LIN {X 0,Y 370.068,Z 490.091,A -85,B 0,C 180,E1 -12871.089,E2 -12871.089} C_VEL
LIN {X 0,Y 369.236,Z 499.209,A -85,B 0,C 180,E1 -12872.728,E2 -12872.728} C_VEL
LIN {X 0,Y 368.632,Z 506.554,A -85,B 0,C 180,E1 -12874.374,E2 -12874.374} C_VEL
LIN {X 0,Y 368.208,Z 512.444,A -85,B 0,C 180,E1 -12876.027,E2 -12876.027} C_VEL
LIN {X 0,Y 367.86,Z 517.099,A -85,B 0,C 180,E1 -12877.686,E2 -12877.686} C_VEL
LIN {X 0,Y 367.581,Z 520.649,A -85,B 0,C 180,E1 -12879.354,E2 -12879.354} C_VEL
LIN {X 0,Y 367.418,Z 523.176,A -85,B 0,C 180,E1 -12881.028,E2 -12881.028} C_VEL
LIN {X 0,Y 367.364,Z 524.704,A -85,B 0,C 180,E1 -12882.662,E2 -12882.662} C_VEL
LIN {X 0,Y 367.283,Z 525.373,A -85,B 0,C 180,E1 -12884.405,E2 -12884.405} C_VEL
LIN {X 0,Y 367.336,Z 525.296,A -85,B 0,C 180,E1 -12885.537,E2 -12885.537} C_VEL
LIN {X 0,Y 367.455,Z 524.256,A -85,B 0,C 180,E1 -12887.304,E2 -12887.304} C_VEL
LIN {X 0,Y 367.684,Z 522.431,A -85,B 0,C 180,E1 -12888.963,E2 -12888.963} C_VEL
LIN {X 0,Y 368.051,Z 519.521,A -85,B 0,C 180,E1 -12890.664,E2 -12890.664} C_VEL
LIN {X 0,Y 368.43,Z 516.667,A -85,B 0,C 180,E1 -12891.919,E2 -12891.919} C_VEL
LIN {X 0,Y 368.033,Z 514.487,A -85,B 0,C 180,E1 -12892.771,E2 -12892.771} C_VEL
LIN {X 0,Y 365.711,Z 510.618,A -85,B 0,C 180,E1 -12894.153,E2 -12894.153} C_VEL
LIN {X 0,Y 363.521,Z 506.158,A -85,B 0,C 180,E1 -12895.502,E2 -12895.502} C_VEL
LIN {X 0,Y 363.329,Z 502.988,A -85,B 0,C 180,E1 -12896.289,E2 -12896.289} C_VEL
LIN {X 0,Y 364.425,Z 495.192,A -85,B 0,C 180,E1 -12897.883,E2 -12897.883} C_VEL
LIN {X 0,Y 365.532,Z 486.293,A -85,B 0,C 180,E1 -12899.36,E2 -12899.36} C_VEL
LIN {X 0,Y 366.817,Z 476.517,A -85,B 0,C 180,E1 -12900.658,E2 -12900.658} C_VEL
LIN {X 0,Y 368.109,Z 465.503,A -85,B 0,C 180,E1 -12901.832,E2 -12901.832} C_VEL
LIN {X 0,Y 369.097,Z 454.561,A -85,B 0,C 180,E1 -12902.761,E2 -12902.761} C_VEL
LIN {X 0,Y 370.067,Z 441.667,A -85,B 0,C 180,E1 -12903.582,E2 -12903.582} C_VEL
LIN {X 0,Y 370.776,Z 428.662,A -85,B 0,C 180,E1 -12904.163,E2 -12904.163} C_VEL
LIN {X 0,Y 371.143,Z 416.945,A -85,B 0,C 180,E1 -12904.494,E2 -12904.494} C_VEL
LIN {X 0,Y 372.737,Z 340.838,A -85,B 0,C 180,E1 -12905.987,E2 -12905.987} C_VEL
LIN {X 0,Y 369.659,Z 327.918,A -85,B 0,C 180,E1 -12906.496,E2 -12906.496} C_VEL
LIN {X 0,Y 364.062,Z 314.904,A -85,B 0,C 180,E1 -12907.224,E2 -12907.224} C_VEL
LIN {X 0,Y 361.901,Z 305.408,A -85,B 0,C 180,E1 -12909.94,E2 -12909.94} C_VEL
LIN {X 0,Y 361.838,Z 305.415,A -85,B 0,C 180,E1 -12912.829,E2 -12912.829} C_VEL
LIN {X 0,Y 361.82,Z 305.414,A -85,B 0,C 180,E1 -12915.947,E2 -12915.947} C_VEL
LIN {X 0,Y 361.838,Z 305.414,A -85,B 0,C 180,E1 -12919.244,E2 -12919.244} C_VEL
LIN {X 0,Y 361.866,Z 305.413,A -85,B 0,C 180,E1 -12922.777,E2 -12922.777} C_VEL
LIN {X 0,Y 361.856,Z 305.41,A -85,B 0,C 180,E1 -12925.72,E2 -12925.72} C_VEL
LIN {X 0,Y 361.876,Z 305.401,A -85,B 0,C 180,E1 -12929.672,E2 -12929.672} C_VEL
LIN {X 0,Y 361.956,Z 305.394,A -85,B 0,C 180,E1 -12933.475,E2 -12933.475} C_VEL
LIN {X 0,Y 361.891,Z 305.4,A -85,B 0,C 180,E1 -12937.145,E2 -12937.145} C_VEL
LIN {X 0,Y 361.922,Z 305.396,A -85,B 0,C 180,E1 -12940.724,E2 -12940.724} C_VEL
LIN {X 0,Y 361.947,Z 305.394,A -85,B 0,C 180,E1 -12944.226,E2 -12944.226} C_VEL
LIN {X 0,Y 362,Z 305.386,A -85,B 0,C 180,E1 -12946.528,E2 -12946.528} C_VEL
LIN {X 0,Y 362.032,Z 305.378,A -85,B 0,C 180,E1 -12949.938,E2 -12949.938} C_VEL
LIN {X 0,Y 362.151,Z 305.373,A -85,B 0,C 180,E1 -12952.192,E2 -12952.192} C_VEL
LIN {X 0,Y 362.117,Z 305.372,A -85,B 0,C 180,E1 -12954.431,E2 -12954.431} C_VEL
LIN {X 0,Y 362.281,Z 305.356,A -85,B 0,C 180,E1 -12957.776,E2 -12957.776} C_VEL
LIN {X 0,Y 362.426,Z 305.33,A -85,B 0,C 180,E1 -12960,E2 -12960} C_VEL
LIN {X 0,Y 362.281,Z 305.352,A -85,B 0,C 180,E1 -12962.224,E2 -12962.224} C_VEL
LIN {X 0,Y 362.171,Z 305.362,A -85,B 0,C 180,E1 -12966.686,E2 -12966.686} C_VEL
LIN {X 0,Y 362.075,Z 305.379,A -85,B 0,C 180,E1 -12968.933,E2 -12968.933} C_VEL
LIN {X 0,Y 361.96,Z 305.389,A -85,B 0,C 180,E1 -12972.332,E2 -12972.332} C_VEL
LIN {X 0,Y 361.963,Z 305.393,A -85,B 0,C 180,E1 -12974.62,E2 -12974.62} C_VEL
LIN {X 0,Y 361.961,Z 305.394,A -85,B 0,C 180,E1 -12978.099,E2 -12978.099} C_VEL
LIN {X 0,Y 361.863,Z 305.401,A -85,B 0,C 180,E1 -12981.655,E2 -12981.655} C_VEL
LIN {X 0,Y 361.928,Z 305.392,A -85,B 0,C 180,E1 -12985.29,E2 -12985.29} C_VEL
LIN {X 0,Y 361.919,Z 305.4,A -85,B 0,C 180,E1 -12987.778,E2 -12987.778} C_VEL
LIN {X 0,Y 361.848,Z 305.412,A -85,B 0,C 180,E1 -12991.285,E2 -12991.285} C_VEL
LIN {X 0,Y 361.855,Z 305.402,A -85,B 0,C 180,E1 -12994.28,E2 -12994.28} C_VEL
LIN {X 0,Y 361.864,Z 305.406,A -85,B 0,C 180,E1 -12997.223,E2 -12997.223} C_VEL
LIN {X 0,Y 361.837,Z 305.409,A -85,B 0,C 180,E1 -13000.755,E2 -13000.755} C_VEL
LIN {X 0,Y 361.819,Z 305.414,A -85,B 0,C 180,E1 -13004.368,E2 -13004.368} C_VEL
LIN {X 0,Y 361.838,Z 305.413,A -85,B 0,C 180,E1 -13007.568,E2 -13007.568} C_VEL
LIN {X 0,Y 361.87,Z 305.399,A -85,B 0,C 180,E1 -13010.974,E2 -13010.974} C_VEL
LIN {X 0,Y 361.876,Z 305.405,A -85,B 0,C 180,E1 -13014.655,E2 -13014.655} C_VEL
LIN {X 0,Y 361.937,Z 305.571,A -85,B 0,C 180,E1 -13018.542,E2 -13018.542} C_VEL
LIN {X 0,Y 364.825,Z 317.71,A -85,B 0,C 180,E1 -13021.834,E2 -13021.834} C_VEL
LIN {X 0,Y 366.693,Z 327.189,A -85,B 0,C 180,E1 -13024.263,E2 -13024.263} C_VEL
LIN {X 0,Y 365.539,Z 339.041,A -85,B 0,C 180,E1 -13026.955,E2 -13026.955} C_VEL
LIN {X 0,Y 369.976,Z 360.901,A -85,B 0,C 180,E1 -13027.767,E2 -13027.767} C_VEL
LIN {X 0,Y 372.124,Z 375.435,A -85,B 0,C 180,E1 -13028.232,E2 -13028.232} C_VEL
LIN {X 0,Y 370.71,Z 446.624,A -85,B 0,C 180,E1 -13029.649,E2 -13029.649} C_VEL
LIN {X 0,Y 370.056,Z 459.471,A -85,B 0,C 180,E1 -13030.082,E2 -13030.082} C_VEL
LIN {X 0,Y 369.035,Z 472.494,A -85,B 0,C 180,E1 -13030.749,E2 -13030.749} C_VEL
LIN {X 0,Y 367.885,Z 484.876,A -85,B 0,C 180,E1 -13031.626,E2 -13031.626} C_VEL
LIN {X 0,Y 366.487,Z 496.517,A -85,B 0,C 180,E1 -13032.708,E2 -13032.708} C_VEL
LIN {X 0,Y 365.196,Z 506.992,A -85,B 0,C 180,E1 -13033.94,E2 -13033.94} C_VEL
LIN {X 0,Y 364.106,Z 516.229,A -85,B 0,C 180,E1 -13035.287,E2 -13035.287} C_VEL
LIN {X 0,Y 362.967,Z 524.926,A -85,B 0,C 180,E1 -13036.849,E2 -13036.849} C_VEL
LIN {X 0,Y 361.882,Z 532.433,A -85,B 0,C 180,E1 -13038.517,E2 -13038.517} C_VEL
LIN {X 0,Y 361.11,Z 539.398,A -85,B 0,C 180,E1 -13040.477,E2 -13040.477} C_VEL
LIN {X 0,Y 360.68,Z 544.02,A -85,B 0,C 180,E1 -13042.16,E2 -13042.16} C_VEL
LIN {X 0,Y 360.424,Z 547.785,A -85,B 0,C 180,E1 -13043.969,E2 -13043.969} C_VEL
LIN {X 0,Y 360.366,Z 550.094,A -85,B 0,C 180,E1 -13045.525,E2 -13045.525} C_VEL
LIN {X 0,Y 360.301,Z 551.286,A -85,B 0,C 180,E1 -13046.645,E2 -13046.645} C_VEL
LIN {X 0,Y 360.358,Z 552.41,A -85,B 0,C 180,E1 -13048.882,E2 -13048.882} C_VEL
LIN {X 0,Y 360.423,Z 552.394,A -85,B 0,C 180,E1 -13049.999,E2 -13049.999} C_VEL
LIN {X 0,Y 360.389,Z 551.981,A -85,B 0,C 180,E1 -13051.117,E2 -13051.117} C_VEL
LIN {X 0,Y 360.327,Z 551.127,A -85,B 0,C 180,E1 -13052.235,E2 -13052.235} C_VEL
LIN {X 0,Y 360.322,Z 549.868,A -85,B 0,C 180,E1 -13053.354,E2 -13053.354} C_VEL
LIN {X 0,Y 360.375,Z 547.185,A -85,B 0,C 180,E1 -13055.034,E2 -13055.034} C_VEL
LIN {X 0,Y 360.497,Z 543.466,A -85,B 0,C 180,E1 -13056.716,E2 -13056.716} C_VEL
LIN {X 0,Y 360.741,Z 538.61,A -85,B 0,C 180,E1 -13058.401,E2 -13058.401} C_VEL
LIN {X 0,Y 361.155,Z 532.469,A -85,B 0,C 180,E1 -13060.086,E2 -13060.086} C_VEL
LIN {X 0,Y 361.774,Z 524.821,A -85,B 0,C 180,E1 -13061.769,E2 -13061.769} C_VEL
LIN {X 0,Y 362.468,Z 516.989,A -85,B 0,C 180,E1 -13063.168,E2 -13063.168} C_VEL
LIN {X 0,Y 363.389,Z 507.414,A -85,B 0,C 180,E1 -13064.561,E2 -13064.561} C_VEL
LIN {X 0,Y 364.251,Z 496.765,A -85,B 0,C 180,E1 -13065.814,E2 -13065.814} C_VEL
LIN {X 0,Y 365.096,Z 486.509,A -85,B 0,C 180,E1 -13066.782,E2 -13066.782} C_VEL
LIN {X 0,Y 366.026,Z 474.401,A -85,B 0,C 180,E1 -13067.674,E2 -13067.674} C_VEL
LIN {X 0,Y 366.831,Z 460.902,A -85,B 0,C 180,E1 -13068.391,E2 -13068.391} C_VEL
LIN {X 0,Y 367.36,Z 448.461,A -85,B 0,C 180,E1 -13068.834,E2 -13068.834} C_VEL
LIN {X 0,Y 368.505,Z 373.288,A -85,B 0,C 180,E1 -13070.322,E2 -13070.322} C_VEL
LIN {X 0,Y 363.871,Z 339.579,A -85,B 0,C 180,E1 -13071.257,E2 -13071.257} C_VEL
LIN {X 0,Y 365.148,Z 323.753,A -85,B 0,C 180,E1 -13074.746,E2 -13074.746} C_VEL
LIN {X 0,Y 364.78,Z 319.672,A -85,B 0,C 180,E1 -13075.692,E2 -13075.692} C_VEL
LIN {X 0,Y 362.332,Z 307.298,A -85,B 0,C 180,E1 -13078.688,E2 -13078.688} C_VEL
LIN {X 0,Y 361.932,Z 305.404,A -85,B 0,C 180,E1 -13079.184,E2 -13079.184} C_VEL
LIN {X 0,Y 361.857,Z 305.407,A -85,B 0,C 180,E1 -13083.369,E2 -13083.369} C_VEL
LIN {X 0,Y 361.863,Z 305.406,A -85,B 0,C 180,E1 -13087.017,E2 -13087.017} C_VEL
LIN {X 0,Y 361.85,Z 305.409,A -85,B 0,C 180,E1 -13089.86,E2 -13089.86} C_VEL
LIN {X 0,Y 361.831,Z 305.412,A -85,B 0,C 180,E1 -13092.828,E2 -13092.828} C_VEL
LIN {X 0,Y 361.814,Z 305.413,A -85,B 0,C 180,E1 -13095.945,E2 -13095.945} C_VEL
LIN {X 0,Y 361.831,Z 305.41,A -85,B 0,C 180,E1 -13099.243,E2 -13099.243} C_VEL
LIN {X 0,Y 361.865,Z 305.411,A -85,B 0,C 180,E1 -13102.775,E2 -13102.775} C_VEL
LIN {X 0,Y 361.849,Z 305.407,A -85,B 0,C 180,E1 -13105.719,E2 -13105.719} C_VEL
LIN {X 0,Y 361.87,Z 305.405,A -85,B 0,C 180,E1 -13109.672,E2 -13109.672} C_VEL
LIN {X 0,Y 361.947,Z 305.397,A -85,B 0,C 180,E1 -13113.474,E2 -13113.474} C_VEL
LIN {X 0,Y 361.882,Z 305.409,A -85,B 0,C 180,E1 -13117.144,E2 -13117.144} C_VEL
LIN {X 0,Y 361.898,Z 305.404,A -85,B 0,C 180,E1 -13120.723,E2 -13120.723} C_VEL
LIN {X 0,Y 361.924,Z 305.403,A -85,B 0,C 180,E1 -13123.066,E2 -13123.066} C_VEL
LIN {X 0,Y 361.99,Z 305.39,A -85,B 0,C 180,E1 -13126.527,E2 -13126.527} C_VEL
LIN {X 0,Y 362.023,Z 305.387,A -85,B 0,C 180,E1 -13129.938,E2 -13129.938} C_VEL
LIN {X 0,Y 362.142,Z 305.371,A -85,B 0,C 180,E1 -13132.192,E2 -13132.192} C_VEL
LIN {X 0,Y 362.108,Z 305.375,A -85,B 0,C 180,E1 -13134.431,E2 -13134.431} C_VEL
LIN {X 0,Y 362.273,Z 305.36,A -85,B 0,C 180,E1 -13137.776,E2 -13137.776} C_VEL
LIN {X 0,Y 362.418,Z 305.34,A -85,B 0,C 180,E1 -13140,E2 -13140} C_VEL
LIN {X 0,Y 362.274,Z 305.356,A -85,B 0,C 180,E1 -13142.224,E2 -13142.224} C_VEL
LIN {X 0,Y 362.126,Z 305.373,A -85,B 0,C 180,E1 -13146.687,E2 -13146.687} C_VEL
LIN {X 0,Y 362.022,Z 305.391,A -85,B 0,C 180,E1 -13150.062,E2 -13150.062} C_VEL
LIN {X 0,Y 361.989,Z 305.395,A -85,B 0,C 180,E1 -13153.899,E2 -13153.899} C_VEL
LIN {X 0,Y 361.959,Z 305.398,A -85,B 0,C 180,E1 -13157.939,E2 -13157.939} C_VEL
LIN {X 0,Y 361.853,Z 305.408,A -85,B 0,C 180,E1 -13161.656,E2 -13161.656} C_VEL
LIN {X 0,Y 361.918,Z 305.399,A -85,B 0,C 180,E1 -13165.291,E2 -13165.291} C_VEL
LIN {X 0,Y 361.91,Z 305.401,A -85,B 0,C 180,E1 -13167.779,E2 -13167.779} C_VEL
LIN {X 0,Y 361.839,Z 305.409,A -85,B 0,C 180,E1 -13171.286,E2 -13171.286} C_VEL
LIN {X 0,Y 361.847,Z 305.411,A -85,B 0,C 180,E1 -13174.281,E2 -13174.281} C_VEL
LIN {X 0,Y 361.853,Z 305.408,A -85,B 0,C 180,E1 -13177.223,E2 -13177.223} C_VEL
LIN {X 0,Y 361.807,Z 305.42,A -85,B 0,C 180,E1 -13180.752,E2 -13180.752} C_VEL
LIN {X 0,Y 361.811,Z 305.414,A -85,B 0,C 180,E1 -13184.37,E2 -13184.37} C_VEL
LIN {X 0,Y 361.825,Z 305.411,A -85,B 0,C 180,E1 -13187.57,E2 -13187.57} C_VEL
LIN {X 0,Y 361.84,Z 305.41,A -85,B 0,C 180,E1 -13191.573,E2 -13191.573} C_VEL
LIN {X 0,Y 361.871,Z 305.407,A -85,B 0,C 180,E1 -13194.657,E2 -13194.657} C_VEL
LIN {X 0,Y 361.835,Z 305.409,A -85,B 0,C 180,E1 -13198.372,E2 -13198.372} C_VEL
LIN {X 0,Y 361.864,Z 305.409,A -85,B 0,C 180,E1 -13200.953,E2 -13200.953} C_VEL
LIN {X 0,Y 361.872,Z 305.405,A -85,B 0,C 180,E1 -13204.707,E2 -13204.707} C_VEL
LIN {X 0,Y 361.86,Z 305.406,A -85,B 0,C 180,E1 -13208.346,E2 -13208.346} C_VEL
LIN {X 0,Y 361.92,Z 305.4,A -85,B 0,C 180,E1 -13212.086,E2 -13212.086} C_VEL
LIN {X 0,Y 361.962,Z 305.397,A -85,B 0,C 180,E1 -13215.381,E2 -13215.381} C_VEL
LIN {X 0,Y 361.961,Z 305.393,A -85,B 0,C 180,E1 -13218.805,E2 -13218.805} C_VEL
LIN {X 0,Y 362.053,Z 305.471,A -85,B 0,C 180,E1 -13220.469,E2 -13220.469} C_VEL
LIN {X 0,Y 363.779,Z 314.771,A -85,B 0,C 180,E1 -13222.852,E2 -13222.852} C_VEL
LIN {X 0,Y 365.738,Z 322.475,A -85,B 0,C 180,E1 -13223.108,E2 -13223.108} C_VEL
LIN {X 0,Y 368.937,Z 339.786,A -85,B 0,C 180,E1 -13223.615,E2 -13223.615} C_VEL
LIN {X 0,Y 367.596,Z 422.045,A -85,B 0,C 180,E1 -13225.237,E2 -13225.237} C_VEL
LIN {X 0,Y 367.117,Z 434.922,A -85,B 0,C 180,E1 -13225.701,E2 -13225.701} C_VEL
LIN {X 0,Y 366.581,Z 446.845,A -85,B 0,C 180,E1 -13226.337,E2 -13226.337} C_VEL
LIN {X 0,Y 365.927,Z 457.563,A -85,B 0,C 180,E1 -13227.097,E2 -13227.097} C_VEL
LIN {X 0,Y 365.136,Z 468.372,A -85,B 0,C 180,E1 -13228.071,E2 -13228.071} C_VEL
LIN {X 0,Y 364.2,Z 479.239,A -85,B 0,C 180,E1 -13229.31,E2 -13229.31} C_VEL
LIN {X 0,Y 363.293,Z 488.125,A -85,B 0,C 180,E1 -13230.555,E2 -13230.555} C_VEL
LIN {X 0,Y 362.544,Z 496.267,A -85,B 0,C 180,E1 -13231.945,E2 -13231.945} C_VEL
LIN {X 0,Y 361.803,Z 504.264,A -85,B 0,C 180,E1 -13233.62,E2 -13233.62} C_VEL
LIN {X 0,Y 361.268,Z 509.686,A -85,B 0,C 180,E1 -13235.023,E2 -13235.023} C_VEL
LIN {X 0,Y 360.921,Z 515.054,A -85,B 0,C 180,E1 -13236.736,E2 -13236.736} C_VEL
LIN {X 0,Y 360.632,Z 519.113,A -85,B 0,C 180,E1 -13238.405,E2 -13238.405} C_VEL
LIN {X 0,Y 360.37,Z 522.189,A -85,B 0,C 180,E1 -13240.11,E2 -13240.11} C_VEL
LIN {X 0,Y 360.33,Z 523.691,A -85,B 0,C 180,E1 -13241.248,E2 -13241.248} C_VEL
LIN {X 0,Y 360.265,Z 524.995,A -85,B 0,C 180,E1 -13242.736,E2 -13242.736} C_VEL
LIN {X 0,Y 360.212,Z 525.671,A -85,B 0,C 180,E1 -13244.694,E2 -13244.694} C_VEL
LIN {X 0,Y 360.259,Z 525.482,A -85,B 0,C 180,E1 -13245.85,E2 -13245.85} C_VEL
LIN {X 0,Y 360.358,Z 524.791,A -85,B 0,C 180,E1 -13247.129,E2 -13247.129} C_VEL
LIN {X 0,Y 360.482,Z 523.855,A -85,B 0,C 180,E1 -13248.177,E2 -13248.177} C_VEL
LIN {X 0,Y 360.667,Z 522.386,A -85,B 0,C 180,E1 -13249.346,E2 -13249.346} C_VEL
LIN {X 0,Y 361.022,Z 519.779,A -85,B 0,C 180,E1 -13250.866,E2 -13250.866} C_VEL
LIN {X 0,Y 361.659,Z 515.042,A -85,B 0,C 180,E1 -13252.871,E2 -13252.871} C_VEL
LIN {X 0,Y 362.568,Z 508.512,A -85,B 0,C 180,E1 -13254.916,E2 -13254.916} C_VEL
LIN {X 0,Y 363.329,Z 502.988,A -85,B 0,C 180,E1 -13256.289,E2 -13256.289} C_VEL
LIN {X 0,Y 363.141,Z 499.632,A -85,B 0,C 180,E1 -13257.058,E2 -13257.058} C_VEL
LIN {X 0,Y 361.072,Z 493.967,A -85,B 0,C 180,E1 -13258.31,E2 -13258.31} C_VEL
LIN {X 0,Y 359.182,Z 487.809,A -85,B 0,C 180,E1 -13259.501,E2 -13259.501} C_VEL
LIN {X 0,Y 359.253,Z 483.577,A -85,B 0,C 180,E1 -13260.16,E2 -13260.16} C_VEL
LIN {X 0,Y 360.561,Z 473.729,A -85,B 0,C 180,E1 -13261.413,E2 -13261.413} C_VEL
LIN {X 0,Y 361.9,Z 461.812,A -85,B 0,C 180,E1 -13262.609,E2 -13262.609} C_VEL
LIN {X 0,Y 362.944,Z 450.384,A -85,B 0,C 180,E1 -13263.503,E2 -13263.503} C_VEL
LIN {X 0,Y 363.793,Z 437.787,A -85,B 0,C 180,E1 -13264.24,E2 -13264.24} C_VEL
LIN {X 0,Y 364.457,Z 424.606,A -85,B 0,C 180,E1 -13264.755,E2 -13264.755} C_VEL
LIN {X 0,Y 365.042,Z 398.79,A -85,B 0,C 180,E1 -13265.32,E2 -13265.32} C_VEL
LIN {X 0,Y 366.313,Z 341.765,A -85,B 0,C 180,E1 -13266.456,E2 -13266.456} C_VEL
LIN {X 0,Y 363.572,Z 330.508,A -85,B 0,C 180,E1 -13266.92,E2 -13266.92} C_VEL
LIN {X 0,Y 356.907,Z 315.178,A -85,B 0,C 180,E1 -13267.82,E2 -13267.82} C_VEL
LIN {X 0,Y 354.827,Z 306.287,A -85,B 0,C 180,E1 -13270.451,E2 -13270.451} C_VEL
LIN {X 0,Y 354.769,Z 306.297,A -85,B 0,C 180,E1 -13273.896,E2 -13273.896} C_VEL
LIN {X 0,Y 354.797,Z 306.291,A -85,B 0,C 180,E1 -13277.663,E2 -13277.663} C_VEL
LIN {X 0,Y 354.817,Z 306.277,A -85,B 0,C 180,E1 -13280.666,E2 -13280.666} C_VEL
LIN {X 0,Y 354.824,Z 306.285,A -85,B 0,C 180,E1 -13284.301,E2 -13284.301} C_VEL
LIN {X 0,Y 354.788,Z 306.29,A -85,B 0,C 180,E1 -13287.667,E2 -13287.667} C_VEL
LIN {X 0,Y 354.871,Z 306.276,A -85,B 0,C 180,E1 -13290.621,E2 -13290.621} C_VEL
LIN {X 0,Y 354.901,Z 306.273,A -85,B 0,C 180,E1 -13294.173,E2 -13294.173} C_VEL
LIN {X 0,Y 354.836,Z 306.282,A -85,B 0,C 180,E1 -13297.894,E2 -13297.894} C_VEL
LIN {X 0,Y 354.924,Z 306.27,A -85,B 0,C 180,E1 -13301.891,E2 -13301.891} C_VEL
LIN {X 0,Y 354.944,Z 306.264,A -85,B 0,C 180,E1 -13305.981,E2 -13305.981} C_VEL
LIN {X 0,Y 354.979,Z 306.259,A -85,B 0,C 180,E1 -13309.736,E2 -13309.736} C_VEL
LIN {X 0,Y 355.114,Z 306.25,A -85,B 0,C 180,E1 -13312.037,E2 -13312.037} C_VEL
LIN {X 0,Y 355.091,Z 306.247,A -85,B 0,C 180,E1 -13314.321,E2 -13314.321} C_VEL
LIN {X 0,Y 355.244,Z 306.232,A -85,B 0,C 180,E1 -13317.732,E2 -13317.732} C_VEL
LIN {X 0,Y 355.375,Z 306.208,A -85,B 0,C 180,E1 -13320,E2 -13320} C_VEL
LIN {X 0,Y 355.244,Z 306.229,A -85,B 0,C 180,E1 -13322.268,E2 -13322.268} C_VEL
LIN {X 0,Y 355.137,Z 306.239,A -85,B 0,C 180,E1 -13326.819,E2 -13326.819} C_VEL
LIN {X 0,Y 355.016,Z 306.258,A -85,B 0,C 180,E1 -13329.112,E2 -13329.112} C_VEL
LIN {X 0,Y 354.921,Z 306.27,A -85,B 0,C 180,E1 -13332.581,E2 -13332.581} C_VEL
LIN {X 0,Y 354.89,Z 306.269,A -85,B 0,C 180,E1 -13336.096,E2 -13336.096} C_VEL
LIN {X 0,Y 354.908,Z 306.276,A -85,B 0,C 180,E1 -13338.472,E2 -13338.472} C_VEL
LIN {X 0,Y 354.818,Z 306.28,A -85,B 0,C 180,E1 -13342.107,E2 -13342.107} C_VEL
LIN {X 0,Y 354.9,Z 306.265,A -85,B 0,C 180,E1 -13345.827,E2 -13345.827} C_VEL
LIN {X 0,Y 354.855,Z 306.272,A -85,B 0,C 180,E1 -13349.678,E2 -13349.678} C_VEL
LIN {X 0,Y 354.808,Z 306.28,A -85,B 0,C 180,E1 -13353.702,E2 -13353.702} C_VEL
LIN {X 0,Y 354.799,Z 306.288,A -85,B 0,C 180,E1 -13356.459,E2 -13356.459} C_VEL
LIN {X 0,Y 354.826,Z 306.286,A -85,B 0,C 180,E1 -13359.424,E2 -13359.424} C_VEL
LIN {X 0,Y 354.79,Z 306.291,A -85,B 0,C 180,E1 -13362.867,E2 -13362.867} C_VEL
LIN {X 0,Y 354.768,Z 306.292,A -85,B 0,C 180,E1 -13366.103,E2 -13366.103} C_VEL
LIN {X 0,Y 354.79,Z 306.293,A -85,B 0,C 180,E1 -13369.179,E2 -13369.179} C_VEL
LIN {X 0,Y 354.809,Z 306.291,A -85,B 0,C 180,E1 -13372.403,E2 -13372.403} C_VEL
LIN {X 0,Y 354.814,Z 306.286,A -85,B 0,C 180,E1 -13374.941,E2 -13374.941} C_VEL
LIN {X 0,Y 354.869,Z 306.451,A -85,B 0,C 180,E1 -13378.035,E2 -13378.035} C_VEL
LIN {X 0,Y 357.633,Z 317.839,A -85,B 0,C 180,E1 -13381.219,E2 -13381.219} C_VEL
LIN {X 0,Y 359.745,Z 328.336,A -85,B 0,C 180,E1 -13383.983,E2 -13383.983} C_VEL
LIN {X 0,Y 359.604,Z 331.955,A -85,B 0,C 180,E1 -13384.844,E2 -13384.844} C_VEL
LIN {X 0,Y 358.872,Z 338.719,A -85,B 0,C 180,E1 -13386.404,E2 -13386.404} C_VEL
LIN {X 0,Y 363.562,Z 361.716,A -85,B 0,C 180,E1 -13387.296,E2 -13387.296} C_VEL
LIN {X 0,Y 365.709,Z 376.184,A -85,B 0,C 180,E1 -13387.775,E2 -13387.775} C_VEL
LIN {X 0,Y 364.171,Z 447.686,A -85,B 0,C 180,E1 -13389.23,E2 -13389.23} C_VEL
LIN {X 0,Y 363.369,Z 461.513,A -85,B 0,C 180,E1 -13389.737,E2 -13389.737} C_VEL
LIN {X 0,Y 362.271,Z 474.46,A -85,B 0,C 180,E1 -13390.448,E2 -13390.448} C_VEL
LIN {X 0,Y 360.966,Z 487,A -85,B 0,C 180,E1 -13391.408,E2 -13391.408} C_VEL
LIN {X 0,Y 359.541,Z 498.198,A -85,B 0,C 180,E1 -13392.51,E2 -13392.51} C_VEL
LIN {X 0,Y 358.236,Z 508.311,A -85,B 0,C 180,E1 -13393.765,E2 -13393.765} C_VEL
LIN {X 0,Y 357.068,Z 517.439,A -85,B 0,C 180,E1 -13395.174,E2 -13395.174} C_VEL
LIN {X 0,Y 355.84,Z 526.358,A -85,B 0,C 180,E1 -13396.871,E2 -13396.871} C_VEL
LIN {X 0,Y 354.753,Z 533.563,A -85,B 0,C 180,E1 -13398.573,E2 -13398.573} C_VEL
LIN {X 0,Y 354.071,Z 539.342,A -85,B 0,C 180,E1 -13400.286,E2 -13400.286} C_VEL
LIN {X 0,Y 353.624,Z 543.914,A -85,B 0,C 180,E1 -13402.002,E2 -13402.002} C_VEL
LIN {X 0,Y 353.318,Z 547.914,A -85,B 0,C 180,E1 -13404.029,E2 -13404.029} C_VEL
LIN {X 0,Y 353.279,Z 549.914,A -85,B 0,C 180,E1 -13405.435,E2 -13405.435} C_VEL
LIN {X 0,Y 353.223,Z 551.071,A -85,B 0,C 180,E1 -13406.577,E2 -13406.577} C_VEL
LIN {X 0,Y 353.259,Z 552.154,A -85,B 0,C 180,E1 -13408.859,E2 -13408.859} C_VEL
LIN {X 0,Y 353.328,Z 552.119,A -85,B 0,C 180,E1 -13409.999,E2 -13409.999} C_VEL
LIN {X 0,Y 353.292,Z 551.675,A -85,B 0,C 180,E1 -13411.139,E2 -13411.139} C_VEL
LIN {X 0,Y 353.243,Z 549.517,A -85,B 0,C 180,E1 -13413.421,E2 -13413.421} C_VEL
LIN {X 0,Y 353.278,Z 546.793,A -85,B 0,C 180,E1 -13415.135,E2 -13415.135} C_VEL
LIN {X 0,Y 353.415,Z 543.03,A -85,B 0,C 180,E1 -13416.852,E2 -13416.852} C_VEL
LIN {X 0,Y 353.679,Z 538.128,A -85,B 0,C 180,E1 -13418.57,E2 -13418.57} C_VEL
LIN {X 0,Y 354.12,Z 531.935,A -85,B 0,C 180,E1 -13420.288,E2 -13420.288} C_VEL
LIN {X 0,Y 354.801,Z 524.222,A -85,B 0,C 180,E1 -13422.003,E2 -13422.003} C_VEL
LIN {X 0,Y 355.506,Z 516.304,A -85,B 0,C 180,E1 -13423.431,E2 -13423.431} C_VEL
LIN {X 0,Y 356.437,Z 506.628,A -85,B 0,C 180,E1 -13424.851,E2 -13424.851} C_VEL
LIN {X 0,Y 357.355,Z 495.865,A -85,B 0,C 180,E1 -13426.127,E2 -13426.127} C_VEL
LIN {X 0,Y 358.235,Z 485.46,A -85,B 0,C 180,E1 -13427.113,E2 -13427.113} C_VEL
LIN {X 0,Y 359.229,Z 473.014,A -85,B 0,C 180,E1 -13428.019,E2 -13428.019} C_VEL
LIN {X 0,Y 360,Z 459.877,A -85,B 0,C 180,E1 -13428.716,E2 -13428.716} C_VEL
LIN {X 0,Y 360.627,Z 446.984,A -85,B 0,C 180,E1 -13429.162,E2 -13429.162} C_VEL
LIN {X 0,Y 361.661,Z 373.758,A -85,B 0,C 180,E1 -13430.633,E2 -13430.633} C_VEL
LIN {X 0,Y 356.94,Z 339.318,A -85,B 0,C 180,E1 -13431.611,E2 -13431.611} C_VEL
LIN {X 0,Y 358.184,Z 324.465,A -85,B 0,C 180,E1 -13434.951,E2 -13434.951} C_VEL
LIN {X 0,Y 357.448,Z 319.009,A -85,B 0,C 180,E1 -13436.255,E2 -13436.255} C_VEL
LIN {X 0,Y 354.876,Z 306.283,A -85,B 0,C 180,E1 -13439.431,E2 -13439.431} C_VEL
LIN {X 0,Y 354.803,Z 306.287,A -85,B 0,C 180,E1 -13443.701,E2 -13443.701} C_VEL
LIN {X 0,Y 354.794,Z 306.291,A -85,B 0,C 180,E1 -13446.458,E2 -13446.458} C_VEL
LIN {X 0,Y 354.82,Z 306.283,A -85,B 0,C 180,E1 -13449.422,E2 -13449.422} C_VEL
LIN {X 0,Y 354.783,Z 306.29,A -85,B 0,C 180,E1 -13452.866,E2 -13452.866} C_VEL
LIN {X 0,Y 354.763,Z 306.293,A -85,B 0,C 180,E1 -13456.103,E2 -13456.103} C_VEL
LIN {X 0,Y 354.783,Z 306.289,A -85,B 0,C 180,E1 -13459.178,E2 -13459.178} C_VEL
LIN {X 0,Y 354.806,Z 306.288,A -85,B 0,C 180,E1 -13462.401,E2 -13462.401} C_VEL
LIN {X 0,Y 354.806,Z 306.289,A -85,B 0,C 180,E1 -13464.94,E2 -13464.94} C_VEL
LIN {X 0,Y 354.808,Z 306.287,A -85,B 0,C 180,E1 -13468.398,E2 -13468.398} C_VEL
LIN {X 0,Y 354.847,Z 306.28,A -85,B 0,C 180,E1 -13471.619,E2 -13471.619} C_VEL
LIN {X 0,Y 354.891,Z 306.274,A -85,B 0,C 180,E1 -13474.172,E2 -13474.172} C_VEL
LIN {X 0,Y 354.826,Z 306.282,A -85,B 0,C 180,E1 -13477.893,E2 -13477.893} C_VEL
LIN {X 0,Y 354.914,Z 306.272,A -85,B 0,C 180,E1 -13481.891,E2 -13481.891} C_VEL
LIN {X 0,Y 354.934,Z 306.27,A -85,B 0,C 180,E1 -13485.981,E2 -13485.981} C_VEL
LIN {X 0,Y 354.969,Z 306.268,A -85,B 0,C 180,E1 -13489.736,E2 -13489.736} C_VEL
LIN {X 0,Y 355.105,Z 306.249,A -85,B 0,C 180,E1 -13492.037,E2 -13492.037} C_VEL
LIN {X 0,Y 355.083,Z 306.251,A -85,B 0,C 180,E1 -13494.321,E2 -13494.321} C_VEL
LIN {X 0,Y 355.236,Z 306.237,A -85,B 0,C 180,E1 -13497.732,E2 -13497.732} C_VEL
LIN {X 0,Y 355.388,Z 306.215,A -85,B 0,C 180,E1 -13500,E2 -13500} C_VEL
LIN {X 0,Y 355.237,Z 306.233,A -85,B 0,C 180,E1 -13502.268,E2 -13502.268} C_VEL
LIN {X 0,Y 355.09,Z 306.249,A -85,B 0,C 180,E1 -13506.82,E2 -13506.82} C_VEL
LIN {X 0,Y 354.969,Z 306.268,A -85,B 0,C 180,E1 -13510.264,E2 -13510.264} C_VEL
LIN {X 0,Y 354.934,Z 306.275,A -85,B 0,C 180,E1 -13514.019,E2 -13514.019} C_VEL
LIN {X 0,Y 354.915,Z 306.278,A -85,B 0,C 180,E1 -13518.109,E2 -13518.109} C_VEL
LIN {X 0,Y 354.807,Z 306.29,A -85,B 0,C 180,E1 -13522.108,E2 -13522.108} C_VEL
LIN {X 0,Y 354.89,Z 306.276,A -85,B 0,C 180,E1 -13525.828,E2 -13525.828} C_VEL
LIN {X 0,Y 354.847,Z 306.28,A -85,B 0,C 180,E1 -13529.679,E2 -13529.679} C_VEL
LIN {X 0,Y 354.8,Z 306.286,A -85,B 0,C 180,E1 -13533.703,E2 -13533.703} C_VEL
LIN {X 0,Y 354.79,Z 306.291,A -85,B 0,C 180,E1 -13536.461,E2 -13536.461} C_VEL
LIN {X 0,Y 354.762,Z 306.291,A -85,B 0,C 180,E1 -13539.414,E2 -13539.414} C_VEL
LIN {X 0,Y 354.78,Z 306.294,A -85,B 0,C 180,E1 -13542.868,E2 -13542.868} C_VEL
LIN {X 0,Y 354.761,Z 306.291,A -85,B 0,C 180,E1 -13546.105,E2 -13546.105} C_VEL
LIN {X 0,Y 354.761,Z 306.295,A -85,B 0,C 180,E1 -13549.177,E2 -13549.177} C_VEL
LIN {X 0,Y 354.797,Z 306.287,A -85,B 0,C 180,E1 -13552.405,E2 -13552.405} C_VEL
LIN {X 0,Y 354.809,Z 306.289,A -85,B 0,C 180,E1 -13554.942,E2 -13554.942} C_VEL
LIN {X 0,Y 354.79,Z 306.287,A -85,B 0,C 180,E1 -13558.406,E2 -13558.406} C_VEL
LIN {X 0,Y 354.794,Z 306.29,A -85,B 0,C 180,E1 -13561.615,E2 -13561.615} C_VEL
LIN {X 0,Y 354.839,Z 306.288,A -85,B 0,C 180,E1 -13565.423,E2 -13565.423} C_VEL
LIN {X 0,Y 354.826,Z 306.285,A -85,B 0,C 180,E1 -13569.114,E2 -13569.114} C_VEL
LIN {X 0,Y 354.88,Z 306.276,A -85,B 0,C 180,E1 -13572.72,E2 -13572.72} C_VEL
LIN {X 0,Y 354.952,Z 306.268,A -85,B 0,C 180,E1 -13576.256,E2 -13576.256} C_VEL
LIN {X 0,Y 355.015,Z 306.415,A -85,B 0,C 180,E1 -13580.242,E2 -13580.242} C_VEL
LIN {X 0,Y 356.578,Z 314.795,A -85,B 0,C 180,E1 -13582.481,E2 -13582.481} C_VEL
LIN {X 0,Y 358.947,Z 323.28,A -85,B 0,C 180,E1 -13582.782,E2 -13582.782} C_VEL
LIN {X 0,Y 362.173,Z 341.135,A -85,B 0,C 180,E1 -13583.315,E2 -13583.315} C_VEL
LIN {X 0,Y 360.763,Z 422.114,A -85,B 0,C 180,E1 -13584.937,E2 -13584.937} C_VEL
LIN {X 0,Y 360.264,Z 435.305,A -85,B 0,C 180,E1 -13585.42,E2 -13585.42} C_VEL
LIN {X 0,Y 359.673,Z 447.787,A -85,B 0,C 180,E1 -13586.104,E2 -13586.104} C_VEL
LIN {X 0,Y 358.934,Z 459.382,A -85,B 0,C 180,E1 -13586.963,E2 -13586.963} C_VEL
LIN {X 0,Y 358.056,Z 470.546,A -85,B 0,C 180,E1 -13588.032,E2 -13588.032} C_VEL
LIN {X 0,Y 357.072,Z 481.082,A -85,B 0,C 180,E1 -13589.296,E2 -13589.296} C_VEL
LIN {X 0,Y 356.178,Z 489.705,A -85,B 0,C 180,E1 -13590.566,E2 -13590.566} C_VEL
LIN {X 0,Y 355.43,Z 497.631,A -85,B 0,C 180,E1 -13591.984,E2 -13591.984} C_VEL
LIN {X 0,Y 354.708,Z 505.387,A -85,B 0,C 180,E1 -13593.693,E2 -13593.693} C_VEL
LIN {X 0,Y 354.166,Z 510.695,A -85,B 0,C 180,E1 -13595.124,E2 -13595.124} C_VEL
LIN {X 0,Y 353.836,Z 515.825,A -85,B 0,C 180,E1 -13596.845,E2 -13596.845} C_VEL
LIN {X 0,Y 353.533,Z 519.821,A -85,B 0,C 180,E1 -13598.575,E2 -13598.575} C_VEL
LIN {X 0,Y 353.259,Z 522.778,A -85,B 0,C 180,E1 -13600.315,E2 -13600.315} C_VEL
LIN {X 0,Y 353.215,Z 524.172,A -85,B 0,C 180,E1 -13601.478,E2 -13601.478} C_VEL
LIN {X 0,Y 353.176,Z 525.29,A -85,B 0,C 180,E1 -13602.819,E2 -13602.819} C_VEL
LIN {X 0,Y 353.117,Z 525.926,A -85,B 0,C 180,E1 -13604.996,E2 -13604.996} C_VEL
LIN {X 0,Y 353.294,Z 525.043,A -85,B 0,C 180,E1 -13607.281,E2 -13607.281} C_VEL
LIN {X 0,Y 353.461,Z 523.895,A -85,B 0,C 180,E1 -13608.551,E2 -13608.551} C_VEL
LIN {X 0,Y 353.829,Z 521.384,A -85,B 0,C 180,E1 -13610.341,E2 -13610.341} C_VEL
LIN {X 0,Y 354.372,Z 517.782,A -85,B 0,C 180,E1 -13612.137,E2 -13612.137} C_VEL
LIN {X 0,Y 355.011,Z 513.034,A -85,B 0,C 180,E1 -13613.918,E2 -13613.918} C_VEL
LIN {X 0,Y 355.922,Z 506.754,A -85,B 0,C 180,E1 -13615.748,E2 -13615.748} C_VEL
LIN {X 0,Y 356.983,Z 499.971,A -85,B 0,C 180,E1 -13617.328,E2 -13617.328} C_VEL
LIN {X 0,Y 358.23,Z 490.836,A -85,B 0,C 180,E1 -13619.05,E2 -13619.05} C_VEL
LIN {X 0,Y 359.253,Z 483.577,A -85,B 0,C 180,E1 -13620.16,E2 -13620.16} C_VEL
LIN {X 0,Y 359.36,Z 479.214,A -85,B 0,C 180,E1 -13620.796,E2 -13620.796} C_VEL
LIN {X 0,Y 357.636,Z 471.983,A -85,B 0,C 180,E1 -13621.85,E2 -13621.85} C_VEL
LIN {X 0,Y 355.771,Z 464.293,A -85,B 0,C 180,E1 -13622.813,E2 -13622.813} C_VEL
LIN {X 0,Y 355.64,Z 459.21,A -85,B 0,C 180,E1 -13623.298,E2 -13623.298} C_VEL
LIN {X 0,Y 356.68,Z 447.695,A -85,B 0,C 180,E1 -13624.15,E2 -13624.15} C_VEL
LIN {X 0,Y 357.534,Z 435.085,A -85,B 0,C 180,E1 -13624.84,E2 -13624.84} C_VEL
LIN {X 0,Y 358.119,Z 422.843,A -85,B 0,C 180,E1 -13625.29,E2 -13625.29} C_VEL
LIN {X 0,Y 360.004,Z 343.236,A -85,B 0,C 180,E1 -13626.928,E2 -13626.928} C_VEL
LIN {X 0,Y 357.634,Z 333.366,A -85,B 0,C 180,E1 -13627.343,E2 -13627.343} C_VEL
LIN {X 0,Y 349.749,Z 315.448,A -85,B 0,C 180,E1 -13628.449,E2 -13628.449} C_VEL
LIN {X 0,Y 347.771,Z 307.168,A -85,B 0,C 180,E1 -13630.933,E2 -13630.933} C_VEL
LIN {X 0,Y 347.725,Z 307.174,A -85,B 0,C 180,E1 -13633.408,E2 -13633.408} C_VEL
LIN {X 0,Y 347.727,Z 307.165,A -85,B 0,C 180,E1 -13636.686,E2 -13636.686} C_VEL
LIN {X 0,Y 347.749,Z 307.16,A -85,B 0,C 180,E1 -13640.173,E2 -13640.173} C_VEL
LIN {X 0,Y 347.764,Z 307.169,A -85,B 0,C 180,E1 -13642.679,E2 -13642.679} C_VEL
LIN {X 0,Y 347.75,Z 307.167,A -85,B 0,C 180,E1 -13645.956,E2 -13645.956} C_VEL
LIN {X 0,Y 347.766,Z 307.159,A -85,B 0,C 180,E1 -13649.653,E2 -13649.653} C_VEL
LIN {X 0,Y 347.853,Z 307.152,A -85,B 0,C 180,E1 -13652.745,E2 -13652.745} C_VEL
LIN {X 0,Y 347.79,Z 307.158,A -85,B 0,C 180,E1 -13656.162,E2 -13656.162} C_VEL
LIN {X 0,Y 347.819,Z 307.154,A -85,B 0,C 180,E1 -13659.91,E2 -13659.91} C_VEL
LIN {X 0,Y 347.868,Z 307.148,A -85,B 0,C 180,E1 -13662.359,E2 -13662.359} C_VEL
LIN {X 0,Y 347.899,Z 307.141,A -85,B 0,C 180,E1 -13665.971,E2 -13665.971} C_VEL
LIN {X 0,Y 347.929,Z 307.139,A -85,B 0,C 180,E1 -13669.526,E2 -13669.526} C_VEL
LIN {X 0,Y 348.106,Z 307.122,A -85,B 0,C 180,E1 -13673.042,E2 -13673.042} C_VEL
LIN {X 0,Y 348.206,Z 307.108,A -85,B 0,C 180,E1 -13677.686,E2 -13677.686} C_VEL
LIN {X 0,Y 348.325,Z 307.086,A -85,B 0,C 180,E1 -13680,E2 -13680} C_VEL
LIN {X 0,Y 348.207,Z 307.106,A -85,B 0,C 180,E1 -13682.313,E2 -13682.313} C_VEL
LIN {X 0,Y 348.105,Z 307.115,A -85,B 0,C 180,E1 -13686.958,E2 -13686.958} C_VEL
LIN {X 0,Y 347.929,Z 307.134,A -85,B 0,C 180,E1 -13690.474,E2 -13690.474} C_VEL
LIN {X 0,Y 347.9,Z 307.149,A -85,B 0,C 180,E1 -13694.15,E2 -13694.15} C_VEL
LIN {X 0,Y 347.893,Z 307.148,A -85,B 0,C 180,E1 -13698.29,E2 -13698.29} C_VEL
LIN {X 0,Y 347.769,Z 307.157,A -85,B 0,C 180,E1 -13701.626,E2 -13701.626} C_VEL
LIN {X 0,Y 347.812,Z 307.151,A -85,B 0,C 180,E1 -13705.108,E2 -13705.108} C_VEL
LIN {X 0,Y 347.812,Z 307.158,A -85,B 0,C 180,E1 -13707.694,E2 -13707.694} C_VEL
LIN {X 0,Y 347.765,Z 307.156,A -85,B 0,C 180,E1 -13710.346,E2 -13710.346} C_VEL
LIN {X 0,Y 347.746,Z 307.16,A -85,B 0,C 180,E1 -13714.464,E2 -13714.464} C_VEL
LIN {X 0,Y 347.775,Z 307.162,A -85,B 0,C 180,E1 -13717.988,E2 -13717.988} C_VEL
LIN {X 0,Y 347.752,Z 307.168,A -85,B 0,C 180,E1 -13721.83,E2 -13721.83} C_VEL
LIN {X 0,Y 347.708,Z 307.175,A -85,B 0,C 180,E1 -13725.027,E2 -13725.027} C_VEL
LIN {X 0,Y 347.752,Z 307.167,A -85,B 0,C 180,E1 -13728.397,E2 -13728.397} C_VEL
LIN {X 0,Y 347.775,Z 307.163,A -85,B 0,C 180,E1 -13732.011,E2 -13732.011} C_VEL
LIN {X 0,Y 347.747,Z 307.172,A -85,B 0,C 180,E1 -13735.536,E2 -13735.536} C_VEL
LIN {X 0,Y 347.775,Z 307.231,A -85,B 0,C 180,E1 -13737.471,E2 -13737.471} C_VEL
LIN {X 0,Y 350.73,Z 319.252,A -85,B 0,C 180,E1 -13740.926,E2 -13740.926} C_VEL
LIN {X 0,Y 352.811,Z 329.479,A -85,B 0,C 180,E1 -13743.689,E2 -13743.689} C_VEL
LIN {X 0,Y 352.938,Z 332.051,A -85,B 0,C 180,E1 -13744.335,E2 -13744.335} C_VEL
LIN {X 0,Y 352.185,Z 338.493,A -85,B 0,C 180,E1 -13745.845,E2 -13745.845} C_VEL
LIN {X 0,Y 357.073,Z 362.092,A -85,B 0,C 180,E1 -13746.787,E2 -13746.787} C_VEL
LIN {X 0,Y 359.319,Z 376.569,A -85,B 0,C 180,E1 -13747.289,E2 -13747.289} C_VEL
LIN {X 0,Y 357.787,Z 446.36,A -85,B 0,C 180,E1 -13748.728,E2 -13748.728} C_VEL
LIN {X 0,Y 356.987,Z 459.826,A -85,B 0,C 180,E1 -13749.207,E2 -13749.207} C_VEL
LIN {X 0,Y 355.862,Z 473.164,A -85,B 0,C 180,E1 -13749.931,E2 -13749.931} C_VEL
LIN {X 0,Y 354.67,Z 484.396,A -85,B 0,C 180,E1 -13750.765,E2 -13750.765} C_VEL
LIN {X 0,Y 353.147,Z 496.019,A -85,B 0,C 180,E1 -13751.883,E2 -13751.883} C_VEL
LIN {X 0,Y 351.728,Z 506.487,A -85,B 0,C 180,E1 -13753.158,E2 -13753.158} C_VEL
LIN {X 0,Y 350.506,Z 514.97,A -85,B 0,C 180,E1 -13754.427,E2 -13754.427} C_VEL
LIN {X 0,Y 349.345,Z 523.723,A -85,B 0,C 180,E1 -13756.029,E2 -13756.029} C_VEL
LIN {X 0,Y 348.088,Z 531.346,A -85,B 0,C 180,E1 -13757.76,E2 -13757.76} C_VEL
LIN {X 0,Y 347.287,Z 537.499,A -85,B 0,C 180,E1 -13759.505,E2 -13759.505} C_VEL
LIN {X 0,Y 346.717,Z 542.406,A -85,B 0,C 180,E1 -13761.255,E2 -13761.255} C_VEL
LIN {X 0,Y 346.344,Z 546.205,A -85,B 0,C 180,E1 -13763.006,E2 -13763.006} C_VEL
LIN {X 0,Y 346.23,Z 548.175,A -85,B 0,C 180,E1 -13764.174,E2 -13764.174} C_VEL
LIN {X 0,Y 346.177,Z 549.737,A -85,B 0,C 180,E1 -13765.341,E2 -13765.341} C_VEL
LIN {X 0,Y 346.147,Z 550.855,A -85,B 0,C 180,E1 -13766.507,E2 -13766.507} C_VEL
LIN {X 0,Y 346.161,Z 551.898,A -85,B 0,C 180,E1 -13768.836,E2 -13768.836} C_VEL
LIN {X 0,Y 346.232,Z 551.844,A -85,B 0,C 180,E1 -13769.999,E2 -13769.999} C_VEL
LIN {X 0,Y 346.194,Z 551.362,A -85,B 0,C 180,E1 -13771.162,E2 -13771.162} C_VEL
LIN {X 0,Y 346.167,Z 549.164,A -85,B 0,C 180,E1 -13773.491,E2 -13773.491} C_VEL
LIN {X 0,Y 346.212,Z 545.867,A -85,B 0,C 180,E1 -13775.528,E2 -13775.528} C_VEL
LIN {X 0,Y 346.433,Z 541.08,A -85,B 0,C 180,E1 -13777.576,E2 -13777.576} C_VEL
LIN {X 0,Y 346.819,Z 534.683,A -85,B 0,C 180,E1 -13779.623,E2 -13779.623} C_VEL
LIN {X 0,Y 347.361,Z 527.703,A -85,B 0,C 180,E1 -13781.376,E2 -13781.376} C_VEL
LIN {X 0,Y 348.282,Z 518.951,A -85,B 0,C 180,E1 -13783.12,E2 -13783.12} C_VEL
LIN {X 0,Y 349.27,Z 508.952,A -85,B 0,C 180,E1 -13784.719,E2 -13784.719} C_VEL
LIN {X 0,Y 350.14,Z 499.096,A -85,B 0,C 180,E1 -13785.99,E2 -13785.99} C_VEL
LIN {X 0,Y 350.977,Z 489.152,A -85,B 0,C 180,E1 -13787.028,E2 -13787.028} C_VEL
LIN {X 0,Y 352.052,Z 476.91,A -85,B 0,C 180,E1 -13788.023,E2 -13788.023} C_VEL
LIN {X 0,Y 352.936,Z 464.083,A -85,B 0,C 180,E1 -13788.803,E2 -13788.803} C_VEL
LIN {X 0,Y 353.599,Z 451.279,A -85,B 0,C 180,E1 -13789.332,E2 -13789.332} C_VEL
LIN {X 0,Y 353.996,Z 434.936,A -85,B 0,C 180,E1 -13789.724,E2 -13789.724} C_VEL
LIN {X 0,Y 354.822,Z 374.346,A -85,B 0,C 180,E1 -13790.952,E2 -13790.952} C_VEL
LIN {X 0,Y 350.01,Z 339.062,A -85,B 0,C 180,E1 -13791.975,E2 -13791.975} C_VEL
LIN {X 0,Y 351.215,Z 324.729,A -85,B 0,C 180,E1 -13795.265,E2 -13795.265} C_VEL
LIN {X 0,Y 349.03,Z 312.75,A -85,B 0,C 180,E1 -13798.251,E2 -13798.251} C_VEL
LIN {X 0,Y 347.834,Z 307.161,A -85,B 0,C 180,E1 -13799.717,E2 -13799.717} C_VEL
LIN {X 0,Y 347.745,Z 307.169,A -85,B 0,C 180,E1 -13804.043,E2 -13804.043} C_VEL
LIN {X 0,Y 347.757,Z 307.163,A -85,B 0,C 180,E1 -13807.32,E2 -13807.32} C_VEL
LIN {X 0,Y 347.728,Z 307.173,A -85,B 0,C 180,E1 -13810.296,E2 -13810.296} C_VEL
LIN {X 0,Y 347.718,Z 307.168,A -85,B 0,C 180,E1 -13813.407,E2 -13813.407} C_VEL
LIN {X 0,Y 347.72,Z 307.172,A -85,B 0,C 180,E1 -13816.685,E2 -13816.685} C_VEL
LIN {X 0,Y 347.741,Z 307.167,A -85,B 0,C 180,E1 -13820.172,E2 -13820.172} C_VEL
LIN {X 0,Y 347.759,Z 307.169,A -85,B 0,C 180,E1 -13822.679,E2 -13822.679} C_VEL
LIN {X 0,Y 347.741,Z 307.165,A -85,B 0,C 180,E1 -13825.955,E2 -13825.955} C_VEL
LIN {X 0,Y 347.764,Z 307.162,A -85,B 0,C 180,E1 -13829.653,E2 -13829.653} C_VEL
LIN {X 0,Y 347.845,Z 307.156,A -85,B 0,C 180,E1 -13832.744,E2 -13832.744} C_VEL
LIN {X 0,Y 347.78,Z 307.16,A -85,B 0,C 180,E1 -13836.161,E2 -13836.161} C_VEL
LIN {X 0,Y 347.804,Z 307.157,A -85,B 0,C 180,E1 -13839.909,E2 -13839.909} C_VEL
LIN {X 0,Y 347.858,Z 307.15,A -85,B 0,C 180,E1 -13842.359,E2 -13842.359} C_VEL
LIN {X 0,Y 347.889,Z 307.147,A -85,B 0,C 180,E1 -13845.97,E2 -13845.97} C_VEL
LIN {X 0,Y 347.92,Z 307.148,A -85,B 0,C 180,E1 -13849.525,E2 -13849.525} C_VEL
LIN {X 0,Y 348.065,Z 307.127,A -85,B 0,C 180,E1 -13851.875,E2 -13851.875} C_VEL
LIN {X 0,Y 348.058,Z 307.126,A -85,B 0,C 180,E1 -13854.206,E2 -13854.206} C_VEL
LIN {X 0,Y 348.198,Z 307.114,A -85,B 0,C 180,E1 -13857.687,E2 -13857.687} C_VEL
LIN {X 0,Y 348.337,Z 307.094,A -85,B 0,C 180,E1 -13860,E2 -13860} C_VEL
LIN {X 0,Y 348.199,Z 307.109,A -85,B 0,C 180,E1 -13862.314,E2 -13862.314} C_VEL
LIN {X 0,Y 348.058,Z 307.125,A -85,B 0,C 180,E1 -13866.959,E2 -13866.959} C_VEL
LIN {X 0,Y 347.919,Z 307.144,A -85,B 0,C 180,E1 -13870.475,E2 -13870.475} C_VEL
LIN {X 0,Y 347.89,Z 307.152,A -85,B 0,C 180,E1 -13874.15,E2 -13874.15} C_VEL
LIN {X 0,Y 347.883,Z 307.152,A -85,B 0,C 180,E1 -13878.291,E2 -13878.291} C_VEL
LIN {X 0,Y 347.759,Z 307.164,A -85,B 0,C 180,E1 -13881.627,E2 -13881.627} C_VEL
LIN {X 0,Y 347.803,Z 307.158,A -85,B 0,C 180,E1 -13885.109,E2 -13885.109} C_VEL
LIN {X 0,Y 347.803,Z 307.158,A -85,B 0,C 180,E1 -13887.695,E2 -13887.695} C_VEL
LIN {X 0,Y 347.757,Z 307.168,A -85,B 0,C 180,E1 -13890.347,E2 -13890.347} C_VEL
LIN {X 0,Y 347.738,Z 307.171,A -85,B 0,C 180,E1 -13894.465,E2 -13894.465} C_VEL
LIN {X 0,Y 347.756,Z 307.164,A -85,B 0,C 180,E1 -13897.987,E2 -13897.987} C_VEL
LIN {X 0,Y 347.738,Z 307.165,A -85,B 0,C 180,E1 -13901.832,E2 -13901.832} C_VEL
LIN {X 0,Y 347.7,Z 307.175,A -85,B 0,C 180,E1 -13905.028,E2 -13905.028} C_VEL
LIN {X 0,Y 347.736,Z 307.167,A -85,B 0,C 180,E1 -13908.4,E2 -13908.4} C_VEL
LIN {X 0,Y 347.753,Z 307.166,A -85,B 0,C 180,E1 -13912.68,E2 -13912.68} C_VEL
LIN {X 0,Y 347.746,Z 307.165,A -85,B 0,C 180,E1 -13915.957,E2 -13915.957} C_VEL
LIN {X 0,Y 347.736,Z 307.168,A -85,B 0,C 180,E1 -13919.652,E2 -13919.652} C_VEL
LIN {X 0,Y 347.736,Z 307.17,A -85,B 0,C 180,E1 -13923.601,E2 -13923.601} C_VEL
LIN {X 0,Y 347.758,Z 307.163,A -85,B 0,C 180,E1 -13926.161,E2 -13926.161} C_VEL
LIN {X 0,Y 347.799,Z 307.16,A -85,B 0,C 180,E1 -13929.91,E2 -13929.91} C_VEL
LIN {X 0,Y 347.832,Z 307.16,A -85,B 0,C 180,E1 -13933.569,E2 -13933.569} C_VEL
LIN {X 0,Y 347.887,Z 307.148,A -85,B 0,C 180,E1 -13937.161,E2 -13937.161} C_VEL
LIN {X 0,Y 347.944,Z 307.24,A -85,B 0,C 180,E1 -13939.968,E2 -13939.968} C_VEL
LIN {X 0,Y 349.458,Z 315.047,A -85,B 0,C 180,E1 -13942.102,E2 -13942.102} C_VEL
LIN {X 0,Y 352.307,Z 324.875,A -85,B 0,C 180,E1 -13942.469,E2 -13942.469} C_VEL
LIN {X 0,Y 355.352,Z 341.3,A -85,B 0,C 180,E1 -13942.975,E2 -13942.975} C_VEL
LIN {X 0,Y 353.943,Z 422.151,A -85,B 0,C 180,E1 -13944.625,E2 -13944.625} C_VEL
LIN {X 0,Y 353.495,Z 434.642,A -85,B 0,C 180,E1 -13945.082,E2 -13945.082} C_VEL
LIN {X 0,Y 352.86,Z 447.148,A -85,B 0,C 180,E1 -13945.764,E2 -13945.764} C_VEL
LIN {X 0,Y 352.162,Z 458.109,A -85,B 0,C 180,E1 -13946.569,E2 -13946.569} C_VEL
LIN {X 0,Y 351.339,Z 468.772,A -85,B 0,C 180,E1 -13947.564,E2 -13947.564} C_VEL
LIN {X 0,Y 350.304,Z 479.682,A -85,B 0,C 180,E1 -13948.851,E2 -13948.851} C_VEL
LIN {X 0,Y 349.256,Z 489.476,A -85,B 0,C 180,E1 -13950.289,E2 -13950.289} C_VEL
LIN {X 0,Y 348.459,Z 497.486,A -85,B 0,C 180,E1 -13951.734,E2 -13951.734} C_VEL
LIN {X 0,Y 347.69,Z 505.344,A -85,B 0,C 180,E1 -13953.477,E2 -13953.477} C_VEL
LIN {X 0,Y 347.064,Z 511.624,A -85,B 0,C 180,E1 -13955.229,E2 -13955.229} C_VEL
LIN {X 0,Y 346.711,Z 516.612,A -85,B 0,C 180,E1 -13956.987,E2 -13956.987} C_VEL
LIN {X 0,Y 346.418,Z 520.478,A -85,B 0,C 180,E1 -13958.753,E2 -13958.753} C_VEL
LIN {X 0,Y 346.15,Z 523.314,A -85,B 0,C 180,E1 -13960.53,E2 -13960.53} C_VEL
LIN {X 0,Y 346.104,Z 524.647,A -85,B 0,C 180,E1 -13961.717,E2 -13961.717} C_VEL
LIN {X 0,Y 346.091,Z 525.582,A -85,B 0,C 180,E1 -13962.908,E2 -13962.908} C_VEL
LIN {X 0,Y 346.036,Z 526.091,A -85,B 0,C 180,E1 -13964.107,E2 -13964.107} C_VEL
LIN {X 0,Y 346.033,Z 526.166,A -85,B 0,C 180,E1 -13965.31,E2 -13965.31} C_VEL
LIN {X 0,Y 346.215,Z 525.306,A -85,B 0,C 180,E1 -13967.43,E2 -13967.43} C_VEL
LIN {X 0,Y 346.452,Z 523.892,A -85,B 0,C 180,E1 -13968.94,E2 -13968.94} C_VEL
LIN {X 0,Y 346.686,Z 522.246,A -85,B 0,C 180,E1 -13970.159,E2 -13970.159} C_VEL
LIN {X 0,Y 347.264,Z 518.887,A -85,B 0,C 180,E1 -13971.988,E2 -13971.988} C_VEL
LIN {X 0,Y 347.912,Z 514.348,A -85,B 0,C 180,E1 -13973.83,E2 -13973.83} C_VEL
LIN {X 0,Y 348.844,Z 508.487,A -85,B 0,C 180,E1 -13975.668,E2 -13975.668} C_VEL
LIN {X 0,Y 350.051,Z 501.005,A -85,B 0,C 180,E1 -13977.502,E2 -13977.502} C_VEL
LIN {X 0,Y 351.21,Z 493.291,A -85,B 0,C 180,E1 -13979.03,E2 -13979.03} C_VEL
LIN {X 0,Y 352.585,Z 483.848,A -85,B 0,C 180,E1 -13980.55,E2 -13980.55} C_VEL
LIN {X 0,Y 353.949,Z 473.672,A -85,B 0,C 180,E1 -13981.865,E2 -13981.865} C_VEL
LIN {X 0,Y 355.245,Z 463.01,A -85,B 0,C 180,E1 -13982.96,E2 -13982.96} C_VEL
LIN {X 0,Y 355.64,Z 459.21,A -85,B 0,C 180,E1 -13983.298,E2 -13983.298} C_VEL
LIN {X 0,Y 355.59,Z 454.025,A -85,B 0,C 180,E1 -13983.752,E2 -13983.752} C_VEL
LIN {X 0,Y 352.838,Z 442.096,A -85,B 0,C 180,E1 -13984.814,E2 -13984.814} C_VEL
LIN {X 0,Y 351.446,Z 434.493,A -85,B 0,C 180,E1 -13985.342,E2 -13985.342} C_VEL
LIN {X 0,Y 351.321,Z 431.199,A -85,B 0,C 180,E1 -13985.502,E2 -13985.502} C_VEL
LIN {X 0,Y 351.872,Z 417.403,A -85,B 0,C 180,E1 -13985.924,E2 -13985.924} C_VEL
LIN {X 0,Y 353.703,Z 344.476,A -85,B 0,C 180,E1 -13987.423,E2 -13987.423} C_VEL
LIN {X 0,Y 351.596,Z 335.979,A -85,B 0,C 180,E1 -13987.797,E2 -13987.797} C_VEL
LIN {X 0,Y 343.986,Z 318.818,A -85,B 0,C 180,E1 -13988.883,E2 -13988.883} C_VEL
LIN {X 0,Y 342.583,Z 315.666,A -85,B 0,C 180,E1 -13989.128,E2 -13989.128} C_VEL
LIN {X 0,Y 340.729,Z 308.043,A -85,B 0,C 180,E1 -13991.537,E2 -13991.537} C_VEL
LIN {X 0,Y 340.643,Z 308.056,A -85,B 0,C 180,E1 -13995.454,E2 -13995.454} C_VEL
LIN {X 0,Y 340.689,Z 308.054,A -85,B 0,C 180,E1 -13998.691,E2 -13998.691} C_VEL
LIN {X 0,Y 340.735,Z 308.038,A -85,B 0,C 180,E1 -14001.773,E2 -14001.773} C_VEL
LIN {X 0,Y 340.725,Z 308.043,A -85,B 0,C 180,E1 -14005.595,E2 -14005.595} C_VEL
LIN {X 0,Y 340.706,Z 308.045,A -85,B 0,C 180,E1 -14008.956,E2 -14008.956} C_VEL
LIN {X 0,Y 340.78,Z 308.035,A -85,B 0,C 180,E1 -14012.474,E2 -14012.474} C_VEL
LIN {X 0,Y 340.758,Z 308.036,A -85,B 0,C 180,E1 -14015.638,E2 -14015.638} C_VEL
LIN {X 0,Y 340.75,Z 308.038,A -85,B 0,C 180,E1 -14019.474,E2 -14019.474} C_VEL
LIN {X 0,Y 340.86,Z 308.022,A -85,B 0,C 180,E1 -14021.984,E2 -14021.984} C_VEL
LIN {X 0,Y 340.871,Z 308.015,A -85,B 0,C 180,E1 -14025.705,E2 -14025.705} C_VEL
LIN {X 0,Y 340.872,Z 308.021,A -85,B 0,C 180,E1 -14029.306,E2 -14029.306} C_VEL
LIN {X 0,Y 341.075,Z 307.997,A -85,B 0,C 180,E1 -14032.898,E2 -14032.898} C_VEL
LIN {X 0,Y 341.168,Z 307.984,A -85,B 0,C 180,E1 -14037.639,E2 -14037.639} C_VEL
LIN {X 0,Y 341.276,Z 307.964,A -85,B 0,C 180,E1 -14040,E2 -14040} C_VEL
LIN {X 0,Y 341.168,Z 307.983,A -85,B 0,C 180,E1 -14042.361,E2 -14042.361} C_VEL
LIN {X 0,Y 341.075,Z 307.99,A -85,B 0,C 180,E1 -14047.102,E2 -14047.102} C_VEL
LIN {X 0,Y 340.871,Z 308.011,A -85,B 0,C 180,E1 -14050.694,E2 -14050.694} C_VEL
LIN {X 0,Y 340.864,Z 308.025,A -85,B 0,C 180,E1 -14054.325,E2 -14054.325} C_VEL
LIN {X 0,Y 340.839,Z 308.029,A -85,B 0,C 180,E1 -14058.467,E2 -14058.467} C_VEL
LIN {X 0,Y 340.719,Z 308.035,A -85,B 0,C 180,E1 -14061.842,E2 -14061.842} C_VEL
LIN {X 0,Y 340.773,Z 308.025,A -85,B 0,C 180,E1 -14065.664,E2 -14065.664} C_VEL
LIN {X 0,Y 340.743,Z 308.04,A -85,B 0,C 180,E1 -14068.32,E2 -14068.32} C_VEL
LIN {X 0,Y 340.705,Z 308.041,A -85,B 0,C 180,E1 -14071.044,E2 -14071.044} C_VEL
LIN {X 0,Y 340.719,Z 308.044,A -85,B 0,C 180,E1 -14075.279,E2 -14075.279} C_VEL
LIN {X 0,Y 340.711,Z 308.042,A -85,B 0,C 180,E1 -14078.386,E2 -14078.386} C_VEL
LIN {X 0,Y 340.7,Z 308.046,A -85,B 0,C 180,E1 -14082.045,E2 -14082.045} C_VEL
LIN {X 0,Y 340.654,Z 308.05,A -85,B 0,C 180,E1 -14086.227,E2 -14086.227} C_VEL
LIN {X 0,Y 340.69,Z 308.043,A -85,B 0,C 180,E1 -14089.753,E2 -14089.753} C_VEL
LIN {X 0,Y 340.707,Z 308.044,A -85,B 0,C 180,E1 -14093.258,E2 -14093.258} C_VEL
LIN {X 0,Y 340.736,Z 308.126,A -85,B 0,C 180,E1 -14096.915,E2 -14096.915} C_VEL
LIN {X 0,Y 343.603,Z 319.54,A -85,B 0,C 180,E1 -14100.304,E2 -14100.304} C_VEL
LIN {X 0,Y 345.889,Z 330.637,A -85,B 0,C 180,E1 -14103.383,E2 -14103.383} C_VEL
LIN {X 0,Y 346.111,Z 333.452,A -85,B 0,C 180,E1 -14104.114,E2 -14104.114} C_VEL
LIN {X 0,Y 345.561,Z 338.136,A -85,B 0,C 180,E1 -14105.242,E2 -14105.242} C_VEL
LIN {X 0,Y 350.8,Z 363.428,A -85,B 0,C 180,E1 -14106.296,E2 -14106.296} C_VEL
LIN {X 0,Y 352.938,Z 377.191,A -85,B 0,C 180,E1 -14106.787,E2 -14106.787} C_VEL
LIN {X 0,Y 351.705,Z 431.772,A -85,B 0,C 180,E1 -14107.918,E2 -14107.918} C_VEL
LIN {X 0,Y 351.187,Z 449.791,A -85,B 0,C 180,E1 -14108.347,E2 -14108.347} C_VEL
LIN {X 0,Y 350.354,Z 461.988,A -85,B 0,C 180,E1 -14108.833,E2 -14108.833} C_VEL
LIN {X 0,Y 349.251,Z 474.081,A -85,B 0,C 180,E1 -14109.534,E2 -14109.534} C_VEL
LIN {X 0,Y 348.009,Z 485.007,A -85,B 0,C 180,E1 -14110.382,E2 -14110.382} C_VEL
LIN {X 0,Y 346.433,Z 496.462,A -85,B 0,C 180,E1 -14111.519,E2 -14111.519} C_VEL
LIN {X 0,Y 344.932,Z 506.801,A -85,B 0,C 180,E1 -14112.816,E2 -14112.816} C_VEL
LIN {X 0,Y 343.579,Z 515.77,A -85,B 0,C 180,E1 -14114.208,E2 -14114.208} C_VEL
LIN {X 0,Y 342.444,Z 523.817,A -85,B 0,C 180,E1 -14115.742,E2 -14115.742} C_VEL
LIN {X 0,Y 341.131,Z 531.366,A -85,B 0,C 180,E1 -14117.506,E2 -14117.506} C_VEL
LIN {X 0,Y 340.301,Z 537.465,A -85,B 0,C 180,E1 -14119.287,E2 -14119.287} C_VEL
LIN {X 0,Y 339.683,Z 542.322,A -85,B 0,C 180,E1 -14121.072,E2 -14121.072} C_VEL
LIN {X 0,Y 339.275,Z 546.075,A -85,B 0,C 180,E1 -14122.86,E2 -14122.86} C_VEL
LIN {X 0,Y 339.136,Z 548.111,A -85,B 0,C 180,E1 -14124.109,E2 -14124.109} C_VEL
LIN {X 0,Y 339.08,Z 549.555,A -85,B 0,C 180,E1 -14125.244,E2 -14125.244} C_VEL
LIN {X 0,Y 339.072,Z 550.64,A -85,B 0,C 180,E1 -14126.434,E2 -14126.434} C_VEL
LIN {X 0,Y 339.062,Z 551.643,A -85,B 0,C 180,E1 -14128.811,E2 -14128.811} C_VEL
LIN {X 0,Y 339.137,Z 551.564,A -85,B 0,C 180,E1 -14129.999,E2 -14129.999} C_VEL
LIN {X 0,Y 339.097,Z 551.045,A -85,B 0,C 180,E1 -14131.187,E2 -14131.187} C_VEL
LIN {X 0,Y 339.092,Z 548.805,A -85,B 0,C 180,E1 -14133.564,E2 -14133.564} C_VEL
LIN {X 0,Y 339.113,Z 545.795,A -85,B 0,C 180,E1 -14135.46,E2 -14135.46} C_VEL
LIN {X 0,Y 339.267,Z 542.136,A -85,B 0,C 180,E1 -14137.139,E2 -14137.139} C_VEL
LIN {X 0,Y 339.57,Z 537.133,A -85,B 0,C 180,E1 -14138.929,E2 -14138.929} C_VEL
LIN {X 0,Y 340.023,Z 530.824,A -85,B 0,C 180,E1 -14140.72,E2 -14140.72} C_VEL
LIN {X 0,Y 340.826,Z 522.924,A -85,B 0,C 180,E1 -14142.503,E2 -14142.503} C_VEL
LIN {X 0,Y 341.651,Z 514.845,A -85,B 0,C 180,E1 -14143.986,E2 -14143.986} C_VEL
LIN {X 0,Y 342.583,Z 504.967,A -85,B 0,C 180,E1 -14145.466,E2 -14145.466} C_VEL
LIN {X 0,Y 343.576,Z 493.94,A -85,B 0,C 180,E1 -14146.793,E2 -14146.793} C_VEL
LIN {X 0,Y 344.637,Z 483.141,A -85,B 0,C 180,E1 -14147.81,E2 -14147.81} C_VEL
LIN {X 0,Y 345.675,Z 470.113,A -85,B 0,C 180,E1 -14148.752,E2 -14148.752} C_VEL
LIN {X 0,Y 346.483,Z 457.646,A -85,B 0,C 180,E1 -14149.398,E2 -14149.398} C_VEL
LIN {X 0,Y 347.053,Z 444.705,A -85,B 0,C 180,E1 -14149.827,E2 -14149.827} C_VEL
LIN {X 0,Y 348.018,Z 374.983,A -85,B 0,C 180,E1 -14151.281,E2 -14151.281} C_VEL
LIN {X 0,Y 343.113,Z 338.857,A -85,B 0,C 180,E1 -14152.338,E2 -14152.338} C_VEL
LIN {X 0,Y 344.248,Z 325.851,A -85,B 0,C 180,E1 -14155.385,E2 -14155.385} C_VEL
LIN {X 0,Y 341.941,Z 313.46,A -85,B 0,C 180,E1 -14158.545,E2 -14158.545} C_VEL
LIN {X 0,Y 340.771,Z 308.04,A -85,B 0,C 180,E1 -14159.997,E2 -14159.997} C_VEL
LIN {X 0,Y 340.72,Z 308.044,A -85,B 0,C 180,E1 -14164.403,E2 -14164.403} C_VEL
LIN {X 0,Y 340.706,Z 308.047,A -85,B 0,C 180,E1 -14168.385,E2 -14168.385} C_VEL
LIN {X 0,Y 340.694,Z 308.046,A -85,B 0,C 180,E1 -14172.044,E2 -14172.044} C_VEL
LIN {X 0,Y 340.647,Z 308.052,A -85,B 0,C 180,E1 -14176.226,E2 -14176.226} C_VEL
LIN {X 0,Y 340.683,Z 308.044,A -85,B 0,C 180,E1 -14179.752,E2 -14179.752} C_VEL
LIN {X 0,Y 340.701,Z 308.043,A -85,B 0,C 180,E1 -14183.258,E2 -14183.258} C_VEL
LIN {X 0,Y 340.688,Z 308.044,A -85,B 0,C 180,E1 -14186.153,E2 -14186.153} C_VEL
LIN {X 0,Y 340.768,Z 308.035,A -85,B 0,C 180,E1 -14190.332,E2 -14190.332} C_VEL
LIN {X 0,Y 340.798,Z 308.036,A -85,B 0,C 180,E1 -14193.019,E2 -14193.019} C_VEL
LIN {X 0,Y 340.72,Z 308.044,A -85,B 0,C 180,E1 -14196.927,E2 -14196.927} C_VEL
LIN {X 0,Y 340.782,Z 308.034,A -85,B 0,C 180,E1 -14200.733,E2 -14200.733} C_VEL
LIN {X 0,Y 340.778,Z 308.038,A -85,B 0,C 180,E1 -14203.218,E2 -14203.218} C_VEL
LIN {X 0,Y 340.835,Z 308.027,A -85,B 0,C 180,E1 -14206.89,E2 -14206.89} C_VEL
LIN {X 0,Y 340.92,Z 308.015,A -85,B 0,C 180,E1 -14210.508,E2 -14210.508} C_VEL
LIN {X 0,Y 341.066,Z 307.997,A -85,B 0,C 180,E1 -14212.898,E2 -14212.898} C_VEL
LIN {X 0,Y 341.16,Z 307.991,A -85,B 0,C 180,E1 -14217.639,E2 -14217.639} C_VEL
LIN {X 0,Y 341.287,Z 307.972,A -85,B 0,C 180,E1 -14220,E2 -14220} C_VEL
LIN {X 0,Y 341.161,Z 307.985,A -85,B 0,C 180,E1 -14222.361,E2 -14222.361} C_VEL
LIN {X 0,Y 341.006,Z 308.004,A -85,B 0,C 180,E1 -14227.103,E2 -14227.103} C_VEL
LIN {X 0,Y 340.862,Z 308.022,A -85,B 0,C 180,E1 -14230.694,E2 -14230.694} C_VEL
LIN {X 0,Y 340.855,Z 308.026,A -85,B 0,C 180,E1 -14234.325,E2 -14234.325} C_VEL
LIN {X 0,Y 340.83,Z 308.029,A -85,B 0,C 180,E1 -14238.467,E2 -14238.467} C_VEL
LIN {X 0,Y 340.71,Z 308.043,A -85,B 0,C 180,E1 -14241.842,E2 -14241.842} C_VEL
LIN {X 0,Y 340.764,Z 308.035,A -85,B 0,C 180,E1 -14245.665,E2 -14245.665} C_VEL
LIN {X 0,Y 340.734,Z 308.043,A -85,B 0,C 180,E1 -14248.32,E2 -14248.32} C_VEL
LIN {X 0,Y 340.697,Z 308.044,A -85,B 0,C 180,E1 -14251.045,E2 -14251.045} C_VEL
LIN {X 0,Y 340.711,Z 308.041,A -85,B 0,C 180,E1 -14255.28,E2 -14255.28} C_VEL
LIN {X 0,Y 340.687,Z 308.047,A -85,B 0,C 180,E1 -14258.384,E2 -14258.384} C_VEL
LIN {X 0,Y 340.688,Z 308.044,A -85,B 0,C 180,E1 -14262.045,E2 -14262.045} C_VEL
LIN {X 0,Y 340.646,Z 308.049,A -85,B 0,C 180,E1 -14266.228,E2 -14266.228} C_VEL
LIN {X 0,Y 340.667,Z 308.05,A -85,B 0,C 180,E1 -14268.689,E2 -14268.689} C_VEL
LIN {X 0,Y 340.715,Z 308.041,A -85,B 0,C 180,E1 -14271.772,E2 -14271.772} C_VEL
LIN {X 0,Y 340.72,Z 308.042,A -85,B 0,C 180,E1 -14275.597,E2 -14275.597} C_VEL
LIN {X 0,Y 340.691,Z 308.047,A -85,B 0,C 180,E1 -14278.956,E2 -14278.956} C_VEL
LIN {X 0,Y 340.709,Z 308.044,A -85,B 0,C 180,E1 -14283.013,E2 -14283.013} C_VEL
LIN {X 0,Y 340.743,Z 308.041,A -85,B 0,C 180,E1 -14285.639,E2 -14285.639} C_VEL
LIN {X 0,Y 340.73,Z 308.044,A -85,B 0,C 180,E1 -14289.474,E2 -14289.474} C_VEL
LIN {X 0,Y 340.792,Z 308.033,A -85,B 0,C 180,E1 -14291.982,E2 -14291.982} C_VEL
LIN {X 0,Y 340.87,Z 308.027,A -85,B 0,C 180,E1 -14295.706,E2 -14295.706} C_VEL
LIN {X 0,Y 340.891,Z 308.041,A -85,B 0,C 180,E1 -14299.683,E2 -14299.683} C_VEL
LIN {X 0,Y 342.362,Z 315.527,A -85,B 0,C 180,E1 -14301.723,E2 -14301.723} C_VEL
LIN {X 0,Y 345.778,Z 326.923,A -85,B 0,C 180,E1 -14302.161,E2 -14302.161} C_VEL
LIN {X 0,Y 348.619,Z 342.681,A -85,B 0,C 180,E1 -14302.653,E2 -14302.653} C_VEL
LIN {X 0,Y 347.075,Z 423.342,A -85,B 0,C 180,E1 -14304.336,E2 -14304.336} C_VEL
LIN {X 0,Y 346.599,Z 436.267,A -85,B 0,C 180,E1 -14304.839,E2 -14304.839} C_VEL
LIN {X 0,Y 345.941,Z 448.527,A -85,B 0,C 180,E1 -14305.54,E2 -14305.54} C_VEL
LIN {X 0,Y 345.087,Z 460.787,A -85,B 0,C 180,E1 -14306.498,E2 -14306.498} C_VEL
LIN {X 0,Y 344.128,Z 472.228,A -85,B 0,C 180,E1 -14307.66,E2 -14307.66} C_VEL
LIN {X 0,Y 343.07,Z 482.572,A -85,B 0,C 180,E1 -14308.974,E2 -14308.974} C_VEL
LIN {X 0,Y 342.138,Z 491.031,A -85,B 0,C 180,E1 -14310.295,E2 -14310.295} C_VEL
LIN {X 0,Y 341.166,Z 500.179,A -85,B 0,C 180,E1 -14312.067,E2 -14312.067} C_VEL
LIN {X 0,Y 340.456,Z 507.542,A -85,B 0,C 180,E1 -14313.848,E2 -14313.848} C_VEL
LIN {X 0,Y 339.968,Z 512.546,A -85,B 0,C 180,E1 -14315.339,E2 -14315.339} C_VEL
LIN {X 0,Y 339.603,Z 517.397,A -85,B 0,C 180,E1 -14317.134,E2 -14317.134} C_VEL
LIN {X 0,Y 339.28,Z 521.137,A -85,B 0,C 180,E1 -14318.938,E2 -14318.938} C_VEL
LIN {X 0,Y 339.052,Z 523.847,A -85,B 0,C 180,E1 -14320.753,E2 -14320.753} C_VEL
LIN {X 0,Y 338.987,Z 525.865,A -85,B 0,C 180,E1 -14322.986,E2 -14322.986} C_VEL
LIN {X 0,Y 338.938,Z 526.39,A -85,B 0,C 180,E1 -14324.409,E2 -14324.409} C_VEL
LIN {X 0,Y 338.951,Z 526.406,A -85,B 0,C 180,E1 -14325.638,E2 -14325.638} C_VEL
LIN {X 0,Y 339.147,Z 525.566,A -85,B 0,C 180,E1 -14327.59,E2 -14327.59} C_VEL
LIN {X 0,Y 339.439,Z 523.888,A -85,B 0,C 180,E1 -14329.347,E2 -14329.347} C_VEL
LIN {X 0,Y 340.017,Z 520.538,A -85,B 0,C 180,E1 -14331.544,E2 -14331.544} C_VEL
LIN {X 0,Y 340.789,Z 515.679,A -85,B 0,C 180,E1 -14333.713,E2 -14333.713} C_VEL
LIN {X 0,Y 341.739,Z 510.098,A -85,B 0,C 180,E1 -14335.587,E2 -14335.587} C_VEL
LIN {X 0,Y 342.892,Z 503.019,A -85,B 0,C 180,E1 -14337.463,E2 -14337.463} C_VEL
LIN {X 0,Y 344.155,Z 495.611,A -85,B 0,C 180,E1 -14339.035,E2 -14339.035} C_VEL
LIN {X 0,Y 345.486,Z 486.744,A -85,B 0,C 180,E1 -14340.568,E2 -14340.568} C_VEL
LIN {X 0,Y 346.977,Z 476.795,A -85,B 0,C 180,E1 -14341.949,E2 -14341.949} C_VEL
LIN {X 0,Y 348.442,Z 465.817,A -85,B 0,C 180,E1 -14343.169,E2 -14343.169} C_VEL
LIN {X 0,Y 349.632,Z 454.454,A -85,B 0,C 180,E1 -14344.165,E2 -14344.165} C_VEL
LIN {X 0,Y 350.664,Z 442.397,A -85,B 0,C 180,E1 -14344.96,E2 -14344.96} C_VEL
LIN {X 0,Y 351.321,Z 431.199,A -85,B 0,C 180,E1 -14345.502,E2 -14345.502} C_VEL
LIN {X 0,Y 350.956,Z 425.511,A -85,B 0,C 180,E1 -14345.76,E2 -14345.76} C_VEL
LIN {X 0,Y 346.471,Z 406.921,A -85,B 0,C 180,E1 -14346.609,E2 -14346.609} C_VEL
LIN {X 0,Y 345.907,Z 401.132,A -85,B 0,C 180,E1 -14346.786,E2 -14346.786} C_VEL
LIN {X 0,Y 347.353,Z 345.319,A -85,B 0,C 180,E1 -14347.954,E2 -14347.954} C_VEL
LIN {X 0,Y 345.519,Z 338.337,A -85,B 0,C 180,E1 -14348.282,E2 -14348.282} C_VEL
LIN {X 0,Y 336.946,Z 319.298,A -85,B 0,C 180,E1 -14349.548,E2 -14349.548} C_VEL
LIN {X 0,Y 335.432,Z 316.013,A -85,B 0,C 180,E1 -14349.804,E2 -14349.804} C_VEL
LIN {X 0,Y 333.668,Z 308.924,A -85,B 0,C 180,E1 -14352.105,E2 -14352.105} C_VEL
LIN {X 0,Y 333.598,Z 308.928,A -85,B 0,C 180,E1 -14355.955,E2 -14355.955} C_VEL
LIN {X 0,Y 333.65,Z 308.925,A -85,B 0,C 180,E1 -14359.315,E2 -14359.315} C_VEL
LIN {X 0,Y 333.667,Z 308.924,A -85,B 0,C 180,E1 -14363.168,E2 -14363.168} C_VEL
LIN {X 0,Y 333.676,Z 308.923,A -85,B 0,C 180,E1 -14365.341,E2 -14365.341} C_VEL
LIN {X 0,Y 333.705,Z 308.91,A -85,B 0,C 180,E1 -14369.71,E2 -14369.71} C_VEL
LIN {X 0,Y 333.745,Z 308.911,A -85,B 0,C 180,E1 -14372.401,E2 -14372.401} C_VEL
LIN {X 0,Y 333.729,Z 308.916,A -85,B 0,C 180,E1 -14375.091,E2 -14375.091} C_VEL
LIN {X 0,Y 333.684,Z 308.92,A -85,B 0,C 180,E1 -14379.019,E2 -14379.019} C_VEL
LIN {X 0,Y 333.796,Z 308.898,A -85,B 0,C 180,E1 -14381.589,E2 -14381.589} C_VEL
LIN {X 0,Y 333.81,Z 308.895,A -85,B 0,C 180,E1 -14385.577,E2 -14385.577} C_VEL
LIN {X 0,Y 333.835,Z 308.9,A -85,B 0,C 180,E1 -14389.078,E2 -14389.078} C_VEL
LIN {X 0,Y 334.025,Z 308.875,A -85,B 0,C 180,E1 -14392.747,E2 -14392.747} C_VEL
LIN {X 0,Y 333.809,Z 308.895,A -85,B 0,C 180,E1 -14395.169,E2 -14395.169} C_VEL
LIN {X 0,Y 334.105,Z 308.863,A -85,B 0,C 180,E1 -14397.589,E2 -14397.589} C_VEL
LIN {X 0,Y 334.228,Z 308.841,A -85,B 0,C 180,E1 -14400,E2 -14400} C_VEL
LIN {X 0,Y 334.106,Z 308.863,A -85,B 0,C 180,E1 -14402.411,E2 -14402.411} C_VEL
LIN {X 0,Y 334.025,Z 308.868,A -85,B 0,C 180,E1 -14407.252,E2 -14407.252} C_VEL
LIN {X 0,Y 333.834,Z 308.886,A -85,B 0,C 180,E1 -14410.922,E2 -14410.922} C_VEL
LIN {X 0,Y 333.81,Z 308.9,A -85,B 0,C 180,E1 -14414.634,E2 -14414.634} C_VEL
LIN {X 0,Y 333.798,Z 308.907,A -85,B 0,C 180,E1 -14418.655,E2 -14418.655} C_VEL
LIN {X 0,Y 333.658,Z 308.917,A -85,B 0,C 180,E1 -14422.281,E2 -14422.281} C_VEL
LIN {X 0,Y 333.737,Z 308.903,A -85,B 0,C 180,E1 -14426.246,E2 -14426.246} C_VEL
LIN {X 0,Y 333.712,Z 308.911,A -85,B 0,C 180,E1 -14428.972,E2 -14428.972} C_VEL
LIN {X 0,Y 333.645,Z 308.925,A -85,B 0,C 180,E1 -14432.587,E2 -14432.587} C_VEL
LIN {X 0,Y 333.677,Z 308.919,A -85,B 0,C 180,E1 -14436.139,E2 -14436.139} C_VEL
LIN {X 0,Y 333.648,Z 308.927,A -85,B 0,C 180,E1 -14439.192,E2 -14439.192} C_VEL
LIN {X 0,Y 333.634,Z 308.926,A -85,B 0,C 180,E1 -14442.5,E2 -14442.5} C_VEL
LIN {X 0,Y 333.598,Z 308.928,A -85,B 0,C 180,E1 -14445.955,E2 -14445.955} C_VEL
LIN {X 0,Y 333.649,Z 308.926,A -85,B 0,C 180,E1 -14449.315,E2 -14449.315} C_VEL
LIN {X 0,Y 333.667,Z 308.922,A -85,B 0,C 180,E1 -14453.168,E2 -14453.168} C_VEL
LIN {X 0,Y 333.691,Z 309.078,A -85,B 0,C 180,E1 -14456.345,E2 -14456.345} C_VEL
LIN {X 0,Y 336.391,Z 319.806,A -85,B 0,C 180,E1 -14459.63,E2 -14459.63} C_VEL
LIN {X 0,Y 338.572,Z 329.739,A -85,B 0,C 180,E1 -14462.492,E2 -14462.492} C_VEL
LIN {X 0,Y 339.319,Z 333.879,A -85,B 0,C 180,E1 -14463.635,E2 -14463.635} C_VEL
LIN {X 0,Y 338.888,Z 337.905,A -85,B 0,C 180,E1 -14464.626,E2 -14464.626} C_VEL
LIN {X 0,Y 344.1,Z 362.445,A -85,B 0,C 180,E1 -14465.69,E2 -14465.69} C_VEL
LIN {X 0,Y 346.618,Z 378.238,A -85,B 0,C 180,E1 -14466.28,E2 -14466.28} C_VEL
LIN {X 0,Y 345.333,Z 431.89,A -85,B 0,C 180,E1 -14467.41,E2 -14467.41} C_VEL
LIN {X 0,Y 344.788,Z 449.77,A -85,B 0,C 180,E1 -14467.845,E2 -14467.845} C_VEL
LIN {X 0,Y 343.928,Z 461.884,A -85,B 0,C 180,E1 -14468.339,E2 -14468.339} C_VEL
LIN {X 0,Y 342.771,Z 473.921,A -85,B 0,C 180,E1 -14469.051,E2 -14469.051} C_VEL
LIN {X 0,Y 341.379,Z 485.611,A -85,B 0,C 180,E1 -14469.985,E2 -14469.985} C_VEL
LIN {X 0,Y 339.747,Z 496.907,A -85,B 0,C 180,E1 -14471.142,E2 -14471.142} C_VEL
LIN {X 0,Y 338.18,Z 507.119,A -85,B 0,C 180,E1 -14472.461,E2 -14472.461} C_VEL
LIN {X 0,Y 336.66,Z 516.477,A -85,B 0,C 180,E1 -14473.973,E2 -14473.973} C_VEL
LIN {X 0,Y 335.324,Z 525.278,A -85,B 0,C 180,E1 -14475.743,E2 -14475.743} C_VEL
LIN {X 0,Y 334.034,Z 532.526,A -85,B 0,C 180,E1 -14477.545,E2 -14477.545} C_VEL
LIN {X 0,Y 333.032,Z 539.178,A -85,B 0,C 180,E1 -14479.666,E2 -14479.666} C_VEL
LIN {X 0,Y 332.477,Z 543.601,A -85,B 0,C 180,E1 -14481.49,E2 -14481.49} C_VEL
LIN {X 0,Y 332.202,Z 545.948,A -85,B 0,C 180,E1 -14482.707,E2 -14482.707} C_VEL
LIN {X 0,Y 332.031,Z 548.217,A -85,B 0,C 180,E1 -14484.175,E2 -14484.175} C_VEL
LIN {X 0,Y 331.997,Z 550.427,A -85,B 0,C 180,E1 -14486.358,E2 -14486.358} C_VEL
LIN {X 0,Y 331.965,Z 551.388,A -85,B 0,C 180,E1 -14488.786,E2 -14488.786} C_VEL
LIN {X 0,Y 332.043,Z 551.276,A -85,B 0,C 180,E1 -14489.999,E2 -14489.999} C_VEL
LIN {X 0,Y 332,Z 550.728,A -85,B 0,C 180,E1 -14491.212,E2 -14491.212} C_VEL
LIN {X 0,Y 332.017,Z 548.447,A -85,B 0,C 180,E1 -14493.64,E2 -14493.64} C_VEL
LIN {X 0,Y 332.017,Z 546.665,A -85,B 0,C 180,E1 -14494.856,E2 -14494.856} C_VEL
LIN {X 0,Y 332.156,Z 543.128,A -85,B 0,C 180,E1 -14496.682,E2 -14496.682} C_VEL
LIN {X 0,Y 332.38,Z 538.462,A -85,B 0,C 180,E1 -14498.511,E2 -14498.511} C_VEL
LIN {X 0,Y 332.929,Z 531.399,A -85,B 0,C 180,E1 -14500.643,E2 -14500.643} C_VEL
LIN {X 0,Y 333.716,Z 523.748,A -85,B 0,C 180,E1 -14502.465,E2 -14502.465} C_VEL
LIN {X 0,Y 334.504,Z 515.9,A -85,B 0,C 180,E1 -14503.981,E2 -14503.981} C_VEL
LIN {X 0,Y 335.48,Z 506.276,A -85,B 0,C 180,E1 -14505.493,E2 -14505.493} C_VEL
LIN {X 0,Y 336.52,Z 495.623,A -85,B 0,C 180,E1 -14506.843,E2 -14506.843} C_VEL
LIN {X 0,Y 337.52,Z 485.34,A -85,B 0,C 180,E1 -14507.885,E2 -14507.885} C_VEL
LIN {X 0,Y 338.554,Z 473.161,A -85,B 0,C 180,E1 -14508.847,E2 -14508.847} C_VEL
LIN {X 0,Y 339.447,Z 459.576,A -85,B 0,C 180,E1 -14509.62,E2 -14509.62} C_VEL
LIN {X 0,Y 340.113,Z 447.011,A -85,B 0,C 180,E1 -14510.091,E2 -14510.091} C_VEL
LIN {X 0,Y 341.341,Z 376.5,A -85,B 0,C 180,E1 -14511.592,E2 -14511.592} C_VEL
LIN {X 0,Y 336.217,Z 338.517,A -85,B 0,C 180,E1 -14512.748,E2 -14512.748} C_VEL
LIN {X 0,Y 337.26,Z 327.875,A -85,B 0,C 180,E1 -14515.288,E2 -14515.288} C_VEL
LIN {X 0,Y 336.201,Z 320.971,A -85,B 0,C 180,E1 -14517.054,E2 -14517.054} C_VEL
LIN {X 0,Y 333.942,Z 310.073,A -85,B 0,C 180,E1 -14519.952,E2 -14519.952} C_VEL
LIN {X 0,Y 333.7,Z 308.92,A -85,B 0,C 180,E1 -14520.289,E2 -14520.289} C_VEL
LIN {X 0,Y 333.671,Z 308.92,A -85,B 0,C 180,E1 -14524.657,E2 -14524.657} C_VEL
LIN {X 0,Y 333.648,Z 308.921,A -85,B 0,C 180,E1 -14527.65,E2 -14527.65} C_VEL
LIN {X 0,Y 333.642,Z 308.924,A -85,B 0,C 180,E1 -14530.766,E2 -14530.766} C_VEL
LIN {X 0,Y 333.589,Z 308.932,A -85,B 0,C 180,E1 -14534.249,E2 -14534.249} C_VEL
LIN {X 0,Y 333.636,Z 308.922,A -85,B 0,C 180,E1 -14537.617,E2 -14537.617} C_VEL
LIN {X 0,Y 333.648,Z 308.922,A -85,B 0,C 180,E1 -14541.201,E2 -14541.201} C_VEL
LIN {X 0,Y 333.671,Z 308.918,A -85,B 0,C 180,E1 -14543.86,E2 -14543.86} C_VEL
LIN {X 0,Y 333.645,Z 308.922,A -85,B 0,C 180,E1 -14547.41,E2 -14547.41} C_VEL
LIN {X 0,Y 333.705,Z 308.918,A -85,B 0,C 180,E1 -14551.027,E2 -14551.027} C_VEL
LIN {X 0,Y 333.728,Z 308.911,A -85,B 0,C 180,E1 -14553.753,E2 -14553.753} C_VEL
LIN {X 0,Y 333.712,Z 308.913,A -85,B 0,C 180,E1 -14557.913,E2 -14557.913} C_VEL
LIN {X 0,Y 333.785,Z 308.904,A -85,B 0,C 180,E1 -14561.589,E2 -14561.589} C_VEL
LIN {X 0,Y 333.8,Z 308.905,A -85,B 0,C 180,E1 -14565.576,E2 -14565.576} C_VEL
LIN {X 0,Y 333.825,Z 308.902,A -85,B 0,C 180,E1 -14569.078,E2 -14569.078} C_VEL
LIN {X 0,Y 334.016,Z 308.874,A -85,B 0,C 180,E1 -14572.747,E2 -14572.747} C_VEL
LIN {X 0,Y 333.801,Z 308.902,A -85,B 0,C 180,E1 -14575.169,E2 -14575.169} C_VEL
LIN {X 0,Y 334.098,Z 308.87,A -85,B 0,C 180,E1 -14577.589,E2 -14577.589} C_VEL
LIN {X 0,Y 334.238,Z 308.85,A -85,B 0,C 180,E1 -14580,E2 -14580} C_VEL
LIN {X 0,Y 334.098,Z 308.865,A -85,B 0,C 180,E1 -14582.411,E2 -14582.411} C_VEL
LIN {X 0,Y 333.96,Z 308.881,A -85,B 0,C 180,E1 -14586.511,E2 -14586.511} C_VEL
LIN {X 0,Y 333.84,Z 308.9,A -85,B 0,C 180,E1 -14589.696,E2 -14589.696} C_VEL
LIN {X 0,Y 333.788,Z 308.904,A -85,B 0,C 180,E1 -14593.392,E2 -14593.392} C_VEL
LIN {X 0,Y 333.739,Z 308.909,A -85,B 0,C 180,E1 -14597.147,E2 -14597.147} C_VEL
LIN {X 0,Y 333.727,Z 308.912,A -85,B 0,C 180,E1 -14599.691,E2 -14599.691} C_VEL
LIN {X 0,Y 333.661,Z 308.919,A -85,B 0,C 180,E1 -14603.591,E2 -14603.591} C_VEL
LIN {X 0,Y 333.728,Z 308.916,A -85,B 0,C 180,E1 -14606.247,E2 -14606.247} C_VEL
LIN {X 0,Y 333.704,Z 308.915,A -85,B 0,C 180,E1 -14608.973,E2 -14608.973} C_VEL
LIN {X 0,Y 333.636,Z 308.927,A -85,B 0,C 180,E1 -14612.588,E2 -14612.588} C_VEL
LIN {X 0,Y 333.669,Z 308.919,A -85,B 0,C 180,E1 -14616.14,E2 -14616.14} C_VEL
LIN {X 0,Y 333.614,Z 308.926,A -85,B 0,C 180,E1 -14619.197,E2 -14619.197} C_VEL
LIN {X 0,Y 333.623,Z 308.927,A -85,B 0,C 180,E1 -14622.5,E2 -14622.5} C_VEL
LIN {X 0,Y 333.591,Z 308.928,A -85,B 0,C 180,E1 -14625.956,E2 -14625.956} C_VEL
LIN {X 0,Y 333.598,Z 308.93,A -85,B 0,C 180,E1 -14629.326,E2 -14629.326} C_VEL
LIN {X 0,Y 333.659,Z 308.925,A -85,B 0,C 180,E1 -14633.17,E2 -14633.17} C_VEL
LIN {X 0,Y 333.671,Z 308.922,A -85,B 0,C 180,E1 -14635.343,E2 -14635.343} C_VEL
LIN {X 0,Y 333.626,Z 308.923,A -85,B 0,C 180,E1 -14638.223,E2 -14638.223} C_VEL
LIN {X 0,Y 333.649,Z 308.924,A -85,B 0,C 180,E1 -14641.023,E2 -14641.023} C_VEL
LIN {X 0,Y 333.694,Z 308.918,A -85,B 0,C 180,E1 -14645.089,E2 -14645.089} C_VEL
LIN {X 0,Y 333.663,Z 308.92,A -85,B 0,C 180,E1 -14649.019,E2 -14649.019} C_VEL
LIN {X 0,Y 333.741,Z 308.915,A -85,B 0,C 180,E1 -14651.588,E2 -14651.588} C_VEL
LIN {X 0,Y 333.809,Z 308.906,A -85,B 0,C 180,E1 -14655.578,E2 -14655.578} C_VEL
LIN {X 0,Y 333.826,Z 308.974,A -85,B 0,C 180,E1 -14659.424,E2 -14659.424} C_VEL
LIN {X 0,Y 335.211,Z 315.798,A -85,B 0,C 180,E1 -14661.316,E2 -14661.316} C_VEL
LIN {X 0,Y 339.237,Z 328.889,A -85,B 0,C 180,E1 -14661.841,E2 -14661.841} C_VEL
LIN {X 0,Y 341.859,Z 344.063,A -85,B 0,C 180,E1 -14662.321,E2 -14662.321} C_VEL
LIN {X 0,Y 340.298,Z 422.825,A -85,B 0,C 180,E1 -14663.987,E2 -14663.987} C_VEL
LIN {X 0,Y 339.796,Z 435.519,A -85,B 0,C 180,E1 -14664.474,E2 -14664.474} C_VEL
LIN {X 0,Y 339.082,Z 448.879,A -85,B 0,C 180,E1 -14665.245,E2 -14665.245} C_VEL
LIN {X 0,Y 338.289,Z 460.201,A -85,B 0,C 180,E1 -14666.137,E2 -14666.137} C_VEL
LIN {X 0,Y 337.284,Z 471.74,A -85,B 0,C 180,E1 -14667.313,E2 -14667.313} C_VEL
LIN {X 0,Y 336.204,Z 482.213,A -85,B 0,C 180,E1 -14668.653,E2 -14668.653} C_VEL
LIN {X 0,Y 335.215,Z 490.785,A -85,B 0,C 180,E1 -14670.001,E2 -14670.001} C_VEL
LIN {X 0,Y 334.379,Z 498.668,A -85,B 0,C 180,E1 -14671.506,E2 -14671.506} C_VEL
LIN {X 0,Y 333.567,Z 506.368,A -85,B 0,C 180,E1 -14673.322,E2 -14673.322} C_VEL
LIN {X 0,Y 332.974,Z 511.648,A -85,B 0,C 180,E1 -14674.844,E2 -14674.844} C_VEL
LIN {X 0,Y 332.604,Z 516.852,A -85,B 0,C 180,E1 -14676.722,E2 -14676.722} C_VEL
LIN {X 0,Y 332.264,Z 520.709,A -85,B 0,C 180,E1 -14678.515,E2 -14678.515} C_VEL
LIN {X 0,Y 332.069,Z 522.755,A -85,B 0,C 180,E1 -14679.749,E2 -14679.749} C_VEL
LIN {X 0,Y 331.962,Z 524.38,A -85,B 0,C 180,E1 -14680.985,E2 -14680.985} C_VEL
LIN {X 0,Y 331.899,Z 526.154,A -85,B 0,C 180,E1 -14683.079,E2 -14683.079} C_VEL
LIN {X 0,Y 331.843,Z 526.689,A -85,B 0,C 180,E1 -14684.724,E2 -14684.724} C_VEL
LIN {X 0,Y 331.883,Z 526.646,A -85,B 0,C 180,E1 -14685.98,E2 -14685.98} C_VEL
LIN {X 0,Y 332.073,Z 525.831,A -85,B 0,C 180,E1 -14687.752,E2 -14687.752} C_VEL
LIN {X 0,Y 332.453,Z 523.89,A -85,B 0,C 180,E1 -14689.77,E2 -14689.77} C_VEL
LIN {X 0,Y 333.029,Z 520.8,A -85,B 0,C 180,E1 -14691.79,E2 -14691.79} C_VEL
LIN {X 0,Y 333.682,Z 516.982,A -85,B 0,C 180,E1 -14693.59,E2 -14693.59} C_VEL
LIN {X 0,Y 334.727,Z 511.075,A -85,B 0,C 180,E1 -14695.698,E2 -14695.698} C_VEL
LIN {X 0,Y 336.028,Z 503.658,A -85,B 0,C 180,E1 -14697.734,E2 -14697.734} C_VEL
LIN {X 0,Y 337.27,Z 496.742,A -85,B 0,C 180,E1 -14699.252,E2 -14699.252} C_VEL
LIN {X 0,Y 338.721,Z 487.596,A -85,B 0,C 180,E1 -14700.9,E2 -14700.9} C_VEL
LIN {X 0,Y 340.21,Z 478.135,A -85,B 0,C 180,E1 -14702.26,E2 -14702.26} C_VEL
LIN {X 0,Y 341.801,Z 466.951,A -85,B 0,C 180,E1 -14703.546,E2 -14703.546} C_VEL
LIN {X 0,Y 343.146,Z 454.886,A -85,B 0,C 180,E1 -14704.636,E2 -14704.636} C_VEL
LIN {X 0,Y 344.228,Z 442.924,A -85,B 0,C 180,E1 -14705.441,E2 -14705.441} C_VEL
LIN {X 0,Y 345.035,Z 430.063,A -85,B 0,C 180,E1 -14706.061,E2 -14706.061} C_VEL
LIN {X 0,Y 345.525,Z 416.875,A -85,B 0,C 180,E1 -14706.454,E2 -14706.454} C_VEL
LIN {X 0,Y 345.907,Z 401.132,A -85,B 0,C 180,E1 -14706.786,E2 -14706.786} C_VEL
LIN {X 0,Y 345.341,Z 395.34,A -85,B 0,C 180,E1 -14706.968,E2 -14706.968} C_VEL
LIN {X 0,Y 340.907,Z 376.664,A -85,B 0,C 180,E1 -14707.797,E2 -14707.797} C_VEL
LIN {X 0,Y 340.506,Z 370.865,A -85,B 0,C 180,E1 -14707.971,E2 -14707.971} C_VEL
LIN {X 0,Y 341.161,Z 346.851,A -85,B 0,C 180,E1 -14708.481,E2 -14708.481} C_VEL
LIN {X 0,Y 339.674,Z 341.257,A -85,B 0,C 180,E1 -14708.754,E2 -14708.754} C_VEL
LIN {X 0,Y 331.603,Z 323.248,A -85,B 0,C 180,E1 -14709.985,E2 -14709.985} C_VEL
LIN {X 0,Y 328.267,Z 316.34,A -85,B 0,C 180,E1 -14710.53,E2 -14710.53} C_VEL
LIN {X 0,Y 326.571,Z 309.807,A -85,B 0,C 180,E1 -14712.703,E2 -14712.703} C_VEL
LIN {X 0,Y 326.578,Z 309.8,A -85,B 0,C 180,E1 -14717.028,E2 -14717.028} C_VEL
LIN {X 0,Y 326.614,Z 309.789,A -85,B 0,C 180,E1 -14720.773,E2 -14720.773} C_VEL
LIN {X 0,Y 326.614,Z 309.799,A -85,B 0,C 180,E1 -14724.48,E2 -14724.48} C_VEL
LIN {X 0,Y 326.61,Z 309.799,A -85,B 0,C 180,E1 -14727.455,E2 -14727.455} C_VEL
LIN {X 0,Y 326.662,Z 309.788,A -85,B 0,C 180,E1 -14730.341,E2 -14730.341} C_VEL
LIN {X 0,Y 326.692,Z 309.788,A -85,B 0,C 180,E1 -14734.516,E2 -14734.516} C_VEL
LIN {X 0,Y 326.649,Z 309.793,A -85,B 0,C 180,E1 -14738.545,E2 -14738.545} C_VEL
LIN {X 0,Y 326.746,Z 309.775,A -85,B 0,C 180,E1 -14741.177,E2 -14741.177} C_VEL
LIN {X 0,Y 326.765,Z 309.772,A -85,B 0,C 180,E1 -14745.433,E2 -14745.433} C_VEL
LIN {X 0,Y 326.771,Z 309.779,A -85,B 0,C 180,E1 -14748.839,E2 -14748.839} C_VEL
LIN {X 0,Y 326.977,Z 309.753,A -85,B 0,C 180,E1 -14752.59,E2 -14752.59} C_VEL
LIN {X 0,Y 326.776,Z 309.772,A -85,B 0,C 180,E1 -14755.065,E2 -14755.065} C_VEL
LIN {X 0,Y 327.046,Z 309.742,A -85,B 0,C 180,E1 -14757.537,E2 -14757.537} C_VEL
LIN {X 0,Y 327.18,Z 309.719,A -85,B 0,C 180,E1 -14760,E2 -14760} C_VEL
LIN {X 0,Y 327.047,Z 309.743,A -85,B 0,C 180,E1 -14762.463,E2 -14762.463} C_VEL
LIN {X 0,Y 326.996,Z 309.74,A -85,B 0,C 180,E1 -14766.169,E2 -14766.169} C_VEL
LIN {X 0,Y 326.916,Z 309.76,A -85,B 0,C 180,E1 -14768.655,E2 -14768.655} C_VEL
LIN {X 0,Y 326.735,Z 309.776,A -85,B 0,C 180,E1 -14772.421,E2 -14772.421} C_VEL
LIN {X 0,Y 326.756,Z 309.776,A -85,B 0,C 180,E1 -14774.957,E2 -14774.957} C_VEL
LIN {X 0,Y 326.734,Z 309.785,A -85,B 0,C 180,E1 -14778.838,E2 -14778.838} C_VEL
LIN {X 0,Y 326.604,Z 309.801,A -85,B 0,C 180,E1 -14782.789,E2 -14782.789} C_VEL
LIN {X 0,Y 326.691,Z 309.779,A -85,B 0,C 180,E1 -14785.484,E2 -14785.484} C_VEL
LIN {X 0,Y 326.662,Z 309.784,A -85,B 0,C 180,E1 -14789.659,E2 -14789.659} C_VEL
LIN {X 0,Y 326.608,Z 309.792,A -85,B 0,C 180,E1 -14794.019,E2 -14794.019} C_VEL
LIN {X 0,Y 326.629,Z 309.793,A -85,B 0,C 180,E1 -14797.238,E2 -14797.238} C_VEL
LIN {X 0,Y 326.579,Z 309.802,A -85,B 0,C 180,E1 -14801.131,E2 -14801.131} C_VEL
LIN {X 0,Y 326.529,Z 309.812,A -85,B 0,C 180,E1 -14804.743,E2 -14804.743} C_VEL
LIN {X 0,Y 326.578,Z 309.803,A -85,B 0,C 180,E1 -14808.154,E2 -14808.154} C_VEL
LIN {X 0,Y 326.6,Z 309.793,A -85,B 0,C 180,E1 -14811.388,E2 -14811.388} C_VEL
LIN {X 0,Y 326.64,Z 309.798,A -85,B 0,C 180,E1 -14815.237,E2 -14815.237} C_VEL
LIN {X 0,Y 326.655,Z 309.907,A -85,B 0,C 180,E1 -14815.706,E2 -14815.706} C_VEL
LIN {X 0,Y 329.444,Z 320.982,A -85,B 0,C 180,E1 -14819.203,E2 -14819.203} C_VEL
LIN {X 0,Y 331.708,Z 331.162,A -85,B 0,C 180,E1 -14822.217,E2 -14822.217} C_VEL
LIN {X 0,Y 332.474,Z 336.273,A -85,B 0,C 180,E1 -14823.646,E2 -14823.646} C_VEL
LIN {X 0,Y 332.277,Z 337.558,A -85,B 0,C 180,E1 -14823.966,E2 -14823.966} C_VEL
LIN {X 0,Y 337.744,Z 362.65,A -85,B 0,C 180,E1 -14825.113,E2 -14825.113} C_VEL
LIN {X 0,Y 340.301,Z 378.74,A -85,B 0,C 180,E1 -14825.732,E2 -14825.732} C_VEL
LIN {X 0,Y 339,Z 432.232,A -85,B 0,C 180,E1 -14826.883,E2 -14826.883} C_VEL
LIN {X 0,Y 338.458,Z 448.761,A -85,B 0,C 180,E1 -14827.288,E2 -14827.288} C_VEL
LIN {X 0,Y 337.524,Z 461.857,A -85,B 0,C 180,E1 -14827.826,E2 -14827.826} C_VEL
LIN {X 0,Y 336.317,Z 473.802,A -85,B 0,C 180,E1 -14828.549,E2 -14828.549} C_VEL
LIN {X 0,Y 334.971,Z 484.668,A -85,B 0,C 180,E1 -14829.425,E2 -14829.425} C_VEL
LIN {X 0,Y 333.273,Z 496.078,A -85,B 0,C 180,E1 -14830.601,E2 -14830.601} C_VEL
LIN {X 0,Y 331.569,Z 506.387,A -85,B 0,C 180,E1 -14831.94,E2 -14831.94} C_VEL
LIN {X 0,Y 329.919,Z 516.189,A -85,B 0,C 180,E1 -14833.544,E2 -14833.544} C_VEL
LIN {X 0,Y 328.44,Z 525.387,A -85,B 0,C 180,E1 -14835.437,E2 -14835.437} C_VEL
LIN {X 0,Y 327.066,Z 532.567,A -85,B 0,C 180,E1 -14837.275,E2 -14837.275} C_VEL
LIN {X 0,Y 326.03,Z 539.135,A -85,B 0,C 180,E1 -14839.441,E2 -14839.441} C_VEL
LIN {X 0,Y 325.417,Z 543.506,A -85,B 0,C 180,E1 -14841.304,E2 -14841.304} C_VEL
LIN {X 0,Y 325.157,Z 545.829,A -85,B 0,C 180,E1 -14842.548,E2 -14842.548} C_VEL
LIN {X 0,Y 324.925,Z 548.29,A -85,B 0,C 180,E1 -14844.248,E2 -14844.248} C_VEL
LIN {X 0,Y 324.901,Z 550.215,A -85,B 0,C 180,E1 -14846.278,E2 -14846.278} C_VEL
LIN {X 0,Y 324.871,Z 551.133,A -85,B 0,C 180,E1 -14848.76,E2 -14848.76} C_VEL
LIN {X 0,Y 324.948,Z 550.979,A -85,B 0,C 180,E1 -14849.999,E2 -14849.999} C_VEL
LIN {X 0,Y 324.904,Z 550.408,A -85,B 0,C 180,E1 -14851.239,E2 -14851.239} C_VEL
LIN {X 0,Y 324.943,Z 548.084,A -85,B 0,C 180,E1 -14853.719,E2 -14853.719} C_VEL
LIN {X 0,Y 325.016,Z 544.566,A -85,B 0,C 180,E1 -14855.91,E2 -14855.91} C_VEL
LIN {X 0,Y 325.225,Z 539.639,A -85,B 0,C 180,E1 -14858.074,E2 -14858.074} C_VEL
LIN {X 0,Y 325.614,Z 534.099,A -85,B 0,C 180,E1 -14859.942,E2 -14859.942} C_VEL
LIN {X 0,Y 326.222,Z 527.161,A -85,B 0,C 180,E1 -14861.809,E2 -14861.809} C_VEL
LIN {X 0,Y 327.068,Z 520.08,A -85,B 0,C 180,E1 -14863.355,E2 -14863.355} C_VEL
LIN {X 0,Y 328.021,Z 511.523,A -85,B 0,C 180,E1 -14864.897,E2 -14864.897} C_VEL
LIN {X 0,Y 329.065,Z 500.911,A -85,B 0,C 180,E1 -14866.437,E2 -14866.437} C_VEL
LIN {X 0,Y 330.062,Z 490.393,A -85,B 0,C 180,E1 -14867.662,E2 -14867.662} C_VEL
LIN {X 0,Y 331.227,Z 478.856,A -85,B 0,C 180,E1 -14868.718,E2 -14868.718} C_VEL
LIN {X 0,Y 332.161,Z 466.881,A -85,B 0,C 180,E1 -14869.545,E2 -14869.545} C_VEL
LIN {X 0,Y 333.015,Z 453.977,A -85,B 0,C 180,E1 -14870.176,E2 -14870.176} C_VEL
LIN {X 0,Y 333.467,Z 440.366,A -85,B 0,C 180,E1 -14870.59,E2 -14870.59} C_VEL
LIN {X 0,Y 334.502,Z 376.572,A -85,B 0,C 180,E1 -14871.957,E2 -14871.957} C_VEL
LIN {X 0,Y 329.307,Z 338.352,A -85,B 0,C 180,E1 -14873.13,E2 -14873.13} C_VEL
LIN {X 0,Y 330.265,Z 328.535,A -85,B 0,C 180,E1 -14875.524,E2 -14875.524} C_VEL
LIN {X 0,Y 328.609,Z 318.908,A -85,B 0,C 180,E1 -14878.066,E2 -14878.066} C_VEL
LIN {X 0,Y 326.629,Z 309.802,A -85,B 0,C 180,E1 -14880.608,E2 -14880.608} C_VEL
LIN {X 0,Y 326.604,Z 309.803,A -85,B 0,C 180,E1 -14884.018,E2 -14884.018} C_VEL
LIN {X 0,Y 326.623,Z 309.796,A -85,B 0,C 180,E1 -14887.237,E2 -14887.237} C_VEL
LIN {X 0,Y 326.573,Z 309.802,A -85,B 0,C 180,E1 -14891.13,E2 -14891.13} C_VEL
LIN {X 0,Y 326.522,Z 309.812,A -85,B 0,C 180,E1 -14894.742,E2 -14894.742} C_VEL
LIN {X 0,Y 326.571,Z 309.805,A -85,B 0,C 180,E1 -14898.153,E2 -14898.153} C_VEL
LIN {X 0,Y 326.618,Z 309.797,A -85,B 0,C 180,E1 -14901.391,E2 -14901.391} C_VEL
LIN {X 0,Y 326.614,Z 309.802,A -85,B 0,C 180,E1 -14904.85,E2 -14904.85} C_VEL
LIN {X 0,Y 326.608,Z 309.798,A -85,B 0,C 180,E1 -14907.456,E2 -14907.456} C_VEL
LIN {X 0,Y 326.655,Z 309.793,A -85,B 0,C 180,E1 -14910.34,E2 -14910.34} C_VEL
LIN {X 0,Y 326.683,Z 309.79,A -85,B 0,C 180,E1 -14914.516,E2 -14914.516} C_VEL
LIN {X 0,Y 326.638,Z 309.795,A -85,B 0,C 180,E1 -14918.545,E2 -14918.545} C_VEL
LIN {X 0,Y 326.736,Z 309.786,A -85,B 0,C 180,E1 -14921.177,E2 -14921.177} C_VEL
LIN {X 0,Y 326.755,Z 309.784,A -85,B 0,C 180,E1 -14925.433,E2 -14925.433} C_VEL
LIN {X 0,Y 326.761,Z 309.78,A -85,B 0,C 180,E1 -14928.839,E2 -14928.839} C_VEL
LIN {X 0,Y 326.97,Z 309.751,A -85,B 0,C 180,E1 -14932.59,E2 -14932.59} C_VEL
LIN {X 0,Y 326.769,Z 309.776,A -85,B 0,C 180,E1 -14935.065,E2 -14935.065} C_VEL
LIN {X 0,Y 327.038,Z 309.748,A -85,B 0,C 180,E1 -14937.537,E2 -14937.537} C_VEL
LIN {X 0,Y 327.189,Z 309.728,A -85,B 0,C 180,E1 -14940,E2 -14940} C_VEL
LIN {X 0,Y 327.039,Z 309.743,A -85,B 0,C 180,E1 -14942.463,E2 -14942.463} C_VEL
LIN {X 0,Y 326.92,Z 309.756,A -85,B 0,C 180,E1 -14946.499,E2 -14946.499} C_VEL
LIN {X 0,Y 326.796,Z 309.779,A -85,B 0,C 180,E1 -14949.907,E2 -14949.907} C_VEL
LIN {X 0,Y 326.751,Z 309.783,A -85,B 0,C 180,E1 -14953.686,E2 -14953.686} C_VEL
LIN {X 0,Y 326.692,Z 309.788,A -85,B 0,C 180,E1 -14957.528,E2 -14957.528} C_VEL
LIN {X 0,Y 326.652,Z 309.798,A -85,B 0,C 180,E1 -14960.136,E2 -14960.136} C_VEL
LIN {X 0,Y 326.641,Z 309.798,A -85,B 0,C 180,E1 -14964.13,E2 -14964.13} C_VEL
LIN {X 0,Y 326.677,Z 309.79,A -85,B 0,C 180,E1 -14966.858,E2 -14966.858} C_VEL
LIN {X 0,Y 326.632,Z 309.799,A -85,B 0,C 180,E1 -14970.612,E2 -14970.612} C_VEL
LIN {X 0,Y 326.6,Z 309.799,A -85,B 0,C 180,E1 -14974.02,E2 -14974.02} C_VEL
LIN {X 0,Y 326.617,Z 309.797,A -85,B 0,C 180,E1 -14977.238,E2 -14977.238} C_VEL
LIN {X 0,Y 326.538,Z 309.809,A -85,B 0,C 180,E1 -14981.126,E2 -14981.126} C_VEL
LIN {X 0,Y 326.555,Z 309.804,A -85,B 0,C 180,E1 -14983.527,E2 -14983.527} C_VEL
LIN {X 0,Y 326.569,Z 309.807,A -85,B 0,C 180,E1 -14987.03,E2 -14987.03} C_VEL
LIN {X 0,Y 326.578,Z 309.804,A -85,B 0,C 180,E1 -14991.387,E2 -14991.387} C_VEL
LIN {X 0,Y 326.616,Z 309.8,A -85,B 0,C 180,E1 -14994.853,E2 -14994.853} C_VEL
LIN {X 0,Y 326.605,Z 309.802,A -85,B 0,C 180,E1 -14997.457,E2 -14997.457} C_VEL
LIN {X 0,Y 326.613,Z 309.797,A -85,B 0,C 180,E1 -15000.338,E2 -15000.338} C_VEL
LIN {X 0,Y 326.639,Z 309.794,A -85,B 0,C 180,E1 -15004.646,E2 -15004.646} C_VEL
LIN {X 0,Y 326.614,Z 309.796,A -85,B 0,C 180,E1 -15008.544,E2 -15008.544} C_VEL
LIN {X 0,Y 326.707,Z 309.788,A -85,B 0,C 180,E1 -15011.176,E2 -15011.176} C_VEL
LIN {X 0,Y 326.764,Z 309.782,A -85,B 0,C 180,E1 -15015.434,E2 -15015.434} C_VEL
LIN {X 0,Y 326.813,Z 309.923,A -85,B 0,C 180,E1 -15019.155,E2 -15019.155} C_VEL
LIN {X 0,Y 328.022,Z 315.81,A -85,B 0,C 180,E1 -15020.878,E2 -15020.878} C_VEL
LIN {X 0,Y 332.637,Z 330.48,A -85,B 0,C 180,E1 -15021.496,E2 -15021.496} C_VEL
LIN {X 0,Y 335.137,Z 345.07,A -85,B 0,C 180,E1 -15021.969,E2 -15021.969} C_VEL
LIN {X 0,Y 333.461,Z 423.627,A -85,B 0,C 180,E1 -15023.667,E2 -15023.667} C_VEL
LIN {X 0,Y 332.928,Z 437.018,A -85,B 0,C 180,E1 -15024.208,E2 -15024.208} C_VEL
LIN {X 0,Y 332.18,Z 450.03,A -85,B 0,C 180,E1 -15024.994,E2 -15024.994} C_VEL
LIN {X 0,Y 331.225,Z 462.657,A -85,B 0,C 180,E1 -15026.051,E2 -15026.051} C_VEL
LIN {X 0,Y 330.195,Z 473.826,A -85,B 0,C 180,E1 -15027.256,E2 -15027.256} C_VEL
LIN {X 0,Y 329.082,Z 483.944,A -85,B 0,C 180,E1 -15028.624,E2 -15028.624} C_VEL
LIN {X 0,Y 327.909,Z 493.887,A -85,B 0,C 180,E1 -15030.308,E2 -15030.308} C_VEL
LIN {X 0,Y 326.941,Z 502.628,A -85,B 0,C 180,E1 -15032.157,E2 -15032.157} C_VEL
LIN {X 0,Y 326.198,Z 509.599,A -85,B 0,C 180,E1 -15034.016,E2 -15034.016} C_VEL
LIN {X 0,Y 325.626,Z 515.99,A -85,B 0,C 180,E1 -15036.196,E2 -15036.196} C_VEL
LIN {X 0,Y 325.249,Z 520.198,A -85,B 0,C 180,E1 -15038.075,E2 -15038.075} C_VEL
LIN {X 0,Y 324.943,Z 523.343,A -85,B 0,C 180,E1 -15039.965,E2 -15039.965} C_VEL
LIN {X 0,Y 324.852,Z 524.903,A -85,B 0,C 180,E1 -15041.229,E2 -15041.229} C_VEL
LIN {X 0,Y 324.815,Z 526.44,A -85,B 0,C 180,E1 -15043.178,E2 -15043.178} C_VEL
LIN {X 0,Y 324.746,Z 526.989,A -85,B 0,C 180,E1 -15045.053,E2 -15045.053} C_VEL
LIN {X 0,Y 324.841,Z 526.859,A -85,B 0,C 180,E1 -15046.336,E2 -15046.336} C_VEL
LIN {X 0,Y 325.014,Z 526.093,A -85,B 0,C 180,E1 -15047.927,E2 -15047.927} C_VEL
LIN {X 0,Y 325.464,Z 523.887,A -85,B 0,C 180,E1 -15050.213,E2 -15050.213} C_VEL
LIN {X 0,Y 326.034,Z 521.076,A -85,B 0,C 180,E1 -15052.041,E2 -15052.041} C_VEL
LIN {X 0,Y 326.826,Z 516.696,A -85,B 0,C 180,E1 -15054.116,E2 -15054.116} C_VEL
LIN {X 0,Y 328.05,Z 510.151,A -85,B 0,C 180,E1 -15056.406,E2 -15056.406} C_VEL
LIN {X 0,Y 329.451,Z 503.044,A -85,B 0,C 180,E1 -15058.328,E2 -15058.328} C_VEL
LIN {X 0,Y 330.791,Z 495.565,A -85,B 0,C 180,E1 -15059.953,E2 -15059.953} C_VEL
LIN {X 0,Y 332.331,Z 486.429,A -85,B 0,C 180,E1 -15061.561,E2 -15061.561} C_VEL
LIN {X 0,Y 333.912,Z 476.635,A -85,B 0,C 180,E1 -15062.951,E2 -15062.951} C_VEL
LIN {X 0,Y 335.57,Z 465.085,A -85,B 0,C 180,E1 -15064.254,E2 -15064.254} C_VEL
LIN {X 0,Y 336.89,Z 453.295,A -85,B 0,C 180,E1 -15065.282,E2 -15065.282} C_VEL
LIN {X 0,Y 338.006,Z 440.782,A -85,B 0,C 180,E1 -15066.101,E2 -15066.101} C_VEL
LIN {X 0,Y 338.786,Z 428.111,A -85,B 0,C 180,E1 -15066.678,E2 -15066.678} C_VEL
LIN {X 0,Y 339.367,Z 412.279,A -85,B 0,C 180,E1 -15067.091,E2 -15067.091} C_VEL
LIN {X 0,Y 340.506,Z 370.865,A -85,B 0,C 180,E1 -15067.971,E2 -15067.971} C_VEL
LIN {X 0,Y 340.198,Z 365.012,A -85,B 0,C 180,E1 -15068.138,E2 -15068.138} C_VEL
LIN {X 0,Y 339.142,Z 359.311,A -85,B 0,C 180,E1 -15068.371,E2 -15068.371} C_VEL
LIN {X 0,Y 338.126,Z 355.618,A -85,B 0,C 180,E1 -15068.555,E2 -15068.555} C_VEL
LIN {X 0,Y 335.57,Z 348.383,A -85,B 0,C 180,E1 -15068.973,E2 -15068.973} C_VEL
LIN {X 0,Y 332.688,Z 341.332,A -85,B 0,C 180,E1 -15069.427,E2 -15069.427} C_VEL
LIN {X 0,Y 324.542,Z 323.627,A -85,B 0,C 180,E1 -15070.718,E2 -15070.718} C_VEL
LIN {X 0,Y 321.069,Z 316.669,A -85,B 0,C 180,E1 -15071.298,E2 -15071.298} C_VEL
LIN {X 0,Y 319.521,Z 310.688,A -85,B 0,C 180,E1 -15073.367,E2 -15073.367} C_VEL
LIN {X 0,Y 319.556,Z 310.674,A -85,B 0,C 180,E1 -15077.017,E2 -15077.017} C_VEL
LIN {X 0,Y 319.549,Z 310.669,A -85,B 0,C 180,E1 -15080.371,E2 -15080.371} C_VEL
LIN {X 0,Y 319.561,Z 310.68,A -85,B 0,C 180,E1 -15083.572,E2 -15083.572} C_VEL
LIN {X 0,Y 319.579,Z 310.674,A -85,B 0,C 180,E1 -15086.687,E2 -15086.687} C_VEL
LIN {X 0,Y 319.593,Z 310.668,A -85,B 0,C 180,E1 -15089.617,E2 -15089.617} C_VEL
LIN {X 0,Y 319.611,Z 310.671,A -85,B 0,C 180,E1 -15092.498,E2 -15092.498} C_VEL
LIN {X 0,Y 319.607,Z 310.674,A -85,B 0,C 180,E1 -15095.304,E2 -15095.304} C_VEL
LIN {X 0,Y 319.599,Z 310.671,A -85,B 0,C 180,E1 -15098.048,E2 -15098.048} C_VEL
LIN {X 0,Y 319.691,Z 310.654,A -85,B 0,C 180,E1 -15100.962,E2 -15100.962} C_VEL
LIN {X 0,Y 319.732,Z 310.648,A -85,B 0,C 180,E1 -15105.276,E2 -15105.276} C_VEL
LIN {X 0,Y 319.759,Z 310.643,A -85,B 0,C 180,E1 -15109.873,E2 -15109.873} C_VEL
LIN {X 0,Y 319.934,Z 310.631,A -85,B 0,C 180,E1 -15112.426,E2 -15112.426} C_VEL
LIN {X 0,Y 319.746,Z 310.648,A -85,B 0,C 180,E1 -15114.956,E2 -15114.956} C_VEL
LIN {X 0,Y 319.99,Z 310.621,A -85,B 0,C 180,E1 -15117.482,E2 -15117.482} C_VEL
LIN {X 0,Y 320.132,Z 310.596,A -85,B 0,C 180,E1 -15120,E2 -15120} C_VEL
LIN {X 0,Y 319.99,Z 310.622,A -85,B 0,C 180,E1 -15122.518,E2 -15122.518} C_VEL
LIN {X 0,Y 319.951,Z 310.617,A -85,B 0,C 180,E1 -15126.305,E2 -15126.305} C_VEL
LIN {X 0,Y 319.844,Z 310.64,A -85,B 0,C 180,E1 -15128.848,E2 -15128.848} C_VEL
LIN {X 0,Y 319.683,Z 310.659,A -85,B 0,C 180,E1 -15132.7,E2 -15132.7} C_VEL
LIN {X 0,Y 319.701,Z 310.653,A -85,B 0,C 180,E1 -15135.295,E2 -15135.295} C_VEL
LIN {X 0,Y 319.675,Z 310.662,A -85,B 0,C 180,E1 -15139.255,E2 -15139.255} C_VEL
LIN {X 0,Y 319.561,Z 310.679,A -85,B 0,C 180,E1 -15143.32,E2 -15143.32} C_VEL
LIN {X 0,Y 319.62,Z 310.66,A -85,B 0,C 180,E1 -15146.089,E2 -15146.089} C_VEL
LIN {X 0,Y 319.591,Z 310.67,A -85,B 0,C 180,E1 -15148.934,E2 -15148.934} C_VEL
LIN {X 0,Y 319.534,Z 310.68,A -85,B 0,C 180,E1 -15151.862,E2 -15151.862} C_VEL
LIN {X 0,Y 319.582,Z 310.677,A -85,B 0,C 180,E1 -15155.543,E2 -15155.543} C_VEL
LIN {X 0,Y 319.559,Z 310.676,A -85,B 0,C 180,E1 -15158.01,E2 -15158.01} C_VEL
LIN {X 0,Y 319.527,Z 310.685,A -85,B 0,C 180,E1 -15161.597,E2 -15161.597} C_VEL
LIN {X 0,Y 319.49,Z 310.688,A -85,B 0,C 180,E1 -15165.257,E2 -15165.257} C_VEL
LIN {X 0,Y 319.53,Z 310.683,A -85,B 0,C 180,E1 -15168.712,E2 -15168.712} C_VEL
LIN {X 0,Y 319.556,Z 310.682,A -85,B 0,C 180,E1 -15172.349,E2 -15172.349} C_VEL
LIN {X 0,Y 319.611,Z 310.78,A -85,B 0,C 180,E1 -15175.046,E2 -15175.046} C_VEL
LIN {X 0,Y 322.554,Z 322.425,A -85,B 0,C 180,E1 -15178.836,E2 -15178.836} C_VEL
LIN {X 0,Y 324.771,Z 332.36,A -85,B 0,C 180,E1 -15181.857,E2 -15181.857} C_VEL
LIN {X 0,Y 325.608,Z 337.257,A -85,B 0,C 180,E1 -15183.273,E2 -15183.273} C_VEL
LIN {X 0,Y 329.237,Z 352.808,A -85,B 0,C 180,E1 -15184.047,E2 -15184.047} C_VEL
LIN {X 0,Y 332.592,Z 370.198,A -85,B 0,C 180,E1 -15184.808,E2 -15184.808} C_VEL
LIN {X 0,Y 334.103,Z 380.201,A -85,B 0,C 180,E1 -15185.195,E2 -15185.195} C_VEL
LIN {X 0,Y 332.29,Z 446.653,A -85,B 0,C 180,E1 -15186.677,E2 -15186.677} C_VEL
LIN {X 0,Y 331.293,Z 460.36,A -85,B 0,C 180,E1 -15187.222,E2 -15187.222} C_VEL
LIN {X 0,Y 330.019,Z 472.708,A -85,B 0,C 180,E1 -15187.954,E2 -15187.954} C_VEL
LIN {X 0,Y 328.619,Z 483.76,A -85,B 0,C 180,E1 -15188.844,E2 -15188.844} C_VEL
LIN {X 0,Y 326.875,Z 495.285,A -85,B 0,C 180,E1 -15190.042,E2 -15190.042} C_VEL
LIN {X 0,Y 325.017,Z 505.688,A -85,B 0,C 180,E1 -15191.4,E2 -15191.4} C_VEL
LIN {X 0,Y 323.396,Z 514.873,A -85,B 0,C 180,E1 -15192.899,E2 -15192.899} C_VEL
LIN {X 0,Y 321.799,Z 524.155,A -85,B 0,C 180,E1 -15194.806,E2 -15194.806} C_VEL
LIN {X 0,Y 320.359,Z 531.499,A -85,B 0,C 180,E1 -15196.682,E2 -15196.682} C_VEL
LIN {X 0,Y 319.296,Z 537.413,A -85,B 0,C 180,E1 -15198.573,E2 -15198.573} C_VEL
LIN {X 0,Y 318.578,Z 542.107,A -85,B 0,C 180,E1 -15200.476,E2 -15200.476} C_VEL
LIN {X 0,Y 318.085,Z 545.71,A -85,B 0,C 180,E1 -15202.381,E2 -15202.381} C_VEL
LIN {X 0,Y 317.844,Z 548.31,A -85,B 0,C 180,E1 -15204.279,E2 -15204.279} C_VEL
LIN {X 0,Y 317.809,Z 550.005,A -85,B 0,C 180,E1 -15206.195,E2 -15206.195} C_VEL
LIN {X 0,Y 317.778,Z 550.634,A -85,B 0,C 180,E1 -15207.464,E2 -15207.464} C_VEL
LIN {X 0,Y 317.78,Z 550.873,A -85,B 0,C 180,E1 -15208.732,E2 -15208.732} C_VEL
LIN {X 0,Y 317.854,Z 550.68,A -85,B 0,C 180,E1 -15209.999,E2 -15209.999} C_VEL
LIN {X 0,Y 317.811,Z 550.087,A -85,B 0,C 180,E1 -15211.266,E2 -15211.266} C_VEL
LIN {X 0,Y 317.8,Z 549.102,A -85,B 0,C 180,E1 -15212.534,E2 -15212.534} C_VEL
LIN {X 0,Y 317.848,Z 547.711,A -85,B 0,C 180,E1 -15213.802,E2 -15213.802} C_VEL
LIN {X 0,Y 317.911,Z 544.524,A -85,B 0,C 180,E1 -15215.84,E2 -15215.84} C_VEL
LIN {X 0,Y 318.06,Z 540.758,A -85,B 0,C 180,E1 -15217.618,E2 -15217.618} C_VEL
LIN {X 0,Y 318.501,Z 534.57,A -85,B 0,C 180,E1 -15219.846,E2 -15219.846} C_VEL
LIN {X 0,Y 319.113,Z 527.797,A -85,B 0,C 180,E1 -15221.753,E2 -15221.753} C_VEL
LIN {X 0,Y 320.095,Z 519.388,A -85,B 0,C 180,E1 -15223.651,E2 -15223.651} C_VEL
LIN {X 0,Y 321.196,Z 509.621,A -85,B 0,C 180,E1 -15225.4,E2 -15225.4} C_VEL
LIN {X 0,Y 322.316,Z 498.789,A -85,B 0,C 180,E1 -15226.955,E2 -15226.955} C_VEL
LIN {X 0,Y 323.309,Z 489.328,A -85,B 0,C 180,E1 -15228.044,E2 -15228.044} C_VEL
LIN {X 0,Y 324.469,Z 477.486,A -85,B 0,C 180,E1 -15229.122,E2 -15229.122} C_VEL
LIN {X 0,Y 325.436,Z 465.146,A -85,B 0,C 180,E1 -15229.966,E2 -15229.966} C_VEL
LIN {X 0,Y 326.24,Z 452.557,A -85,B 0,C 180,E1 -15230.572,E2 -15230.572} C_VEL
LIN {X 0,Y 326.672,Z 439.647,A -85,B 0,C 180,E1 -15230.956,E2 -15230.956} C_VEL
LIN {X 0,Y 327.765,Z 377.515,A -85,B 0,C 180,E1 -15232.312,E2 -15232.312} C_VEL
LIN {X 0,Y 322.415,Z 338.131,A -85,B 0,C 180,E1 -15233.541,E2 -15233.541} C_VEL
LIN {X 0,Y 323.248,Z 329.195,A -85,B 0,C 180,E1 -15235.774,E2 -15235.774} C_VEL
LIN {X 0,Y 321.212,Z 318.159,A -85,B 0,C 180,E1 -15238.772,E2 -15238.772} C_VEL
LIN {X 0,Y 319.567,Z 310.681,A -85,B 0,C 180,E1 -15240.941,E2 -15240.941} C_VEL
LIN {X 0,Y 319.557,Z 310.677,A -85,B 0,C 180,E1 -15244.875,E2 -15244.875} C_VEL
LIN {X 0,Y 319.569,Z 310.678,A -85,B 0,C 180,E1 -15248.007,E2 -15248.007} C_VEL
LIN {X 0,Y 319.521,Z 310.681,A -85,B 0,C 180,E1 -15251.596,E2 -15251.596} C_VEL
LIN {X 0,Y 319.483,Z 310.686,A -85,B 0,C 180,E1 -15255.256,E2 -15255.256} C_VEL
LIN {X 0,Y 319.523,Z 310.684,A -85,B 0,C 180,E1 -15258.711,E2 -15258.711} C_VEL
LIN {X 0,Y 319.572,Z 310.677,A -85,B 0,C 180,E1 -15262.343,E2 -15262.343} C_VEL
LIN {X 0,Y 319.554,Z 310.679,A -85,B 0,C 180,E1 -15265.123,E2 -15265.123} C_VEL
LIN {X 0,Y 319.568,Z 310.679,A -85,B 0,C 180,E1 -15269.056,E2 -15269.056} C_VEL
LIN {X 0,Y 319.602,Z 310.672,A -85,B 0,C 180,E1 -15272.497,E2 -15272.497} C_VEL
LIN {X 0,Y 319.597,Z 310.674,A -85,B 0,C 180,E1 -15275.303,E2 -15275.303} C_VEL
LIN {X 0,Y 319.589,Z 310.672,A -85,B 0,C 180,E1 -15278.047,E2 -15278.047} C_VEL
LIN {X 0,Y 319.681,Z 310.664,A -85,B 0,C 180,E1 -15280.962,E2 -15280.962} C_VEL
LIN {X 0,Y 319.722,Z 310.659,A -85,B 0,C 180,E1 -15285.276,E2 -15285.276} C_VEL
LIN {X 0,Y 319.749,Z 310.653,A -85,B 0,C 180,E1 -15289.873,E2 -15289.873} C_VEL
LIN {X 0,Y 319.924,Z 310.628,A -85,B 0,C 180,E1 -15292.426,E2 -15292.426} C_VEL
LIN {X 0,Y 319.738,Z 310.65,A -85,B 0,C 180,E1 -15294.956,E2 -15294.956} C_VEL
LIN {X 0,Y 319.982,Z 310.626,A -85,B 0,C 180,E1 -15297.482,E2 -15297.482} C_VEL
LIN {X 0,Y 320.141,Z 310.606,A -85,B 0,C 180,E1 -15300,E2 -15300} C_VEL
LIN {X 0,Y 319.982,Z 310.622,A -85,B 0,C 180,E1 -15302.518,E2 -15302.518} C_VEL
LIN {X 0,Y 319.886,Z 310.632,A -85,B 0,C 180,E1 -15306.484,E2 -15306.484} C_VEL
LIN {X 0,Y 319.743,Z 310.657,A -85,B 0,C 180,E1 -15310.128,E2 -15310.128} C_VEL
LIN {X 0,Y 319.723,Z 310.655,A -85,B 0,C 180,E1 -15314.725,E2 -15314.725} C_VEL
LIN {X 0,Y 319.681,Z 310.661,A -85,B 0,C 180,E1 -15319.038,E2 -15319.038} C_VEL
LIN {X 0,Y 319.552,Z 310.676,A -85,B 0,C 180,E1 -15323.321,E2 -15323.321} C_VEL
LIN {X 0,Y 319.627,Z 310.671,A -85,B 0,C 180,E1 -15326.089,E2 -15326.089} C_VEL
LIN {X 0,Y 319.582,Z 310.674,A -85,B 0,C 180,E1 -15328.935,E2 -15328.935} C_VEL
LIN {X 0,Y 319.525,Z 310.68,A -85,B 0,C 180,E1 -15331.863,E2 -15331.863} C_VEL
LIN {X 0,Y 319.573,Z 310.674,A -85,B 0,C 180,E1 -15335.544,E2 -15335.544} C_VEL
LIN {X 0,Y 319.522,Z 310.68,A -85,B 0,C 180,E1 -15339.663,E2 -15339.663} C_VEL
LIN {X 0,Y 319.515,Z 310.681,A -85,B 0,C 180,E1 -15343.461,E2 -15343.461} C_VEL
LIN {X 0,Y 319.547,Z 310.682,A -85,B 0,C 180,E1 -15347.017,E2 -15347.017} C_VEL
LIN {X 0,Y 319.541,Z 310.679,A -85,B 0,C 180,E1 -15350.372,E2 -15350.372} C_VEL
LIN {X 0,Y 319.576,Z 310.674,A -85,B 0,C 180,E1 -15354.459,E2 -15354.459} C_VEL
LIN {X 0,Y 319.521,Z 310.681,A -85,B 0,C 180,E1 -15358.139,E2 -15358.139} C_VEL
LIN {X 0,Y 319.567,Z 310.678,A -85,B 0,C 180,E1 -15361.606,E2 -15361.606} C_VEL
LIN {X 0,Y 319.571,Z 310.68,A -85,B 0,C 180,E1 -15365.303,E2 -15365.303} C_VEL
LIN {X 0,Y 319.565,Z 310.676,A -85,B 0,C 180,E1 -15368.047,E2 -15368.047} C_VEL
LIN {X 0,Y 319.624,Z 310.67,A -85,B 0,C 180,E1 -15372.072,E2 -15372.072} C_VEL
LIN {X 0,Y 319.732,Z 310.656,A -85,B 0,C 180,E1 -15376.009,E2 -15376.009} C_VEL
LIN {X 0,Y 319.737,Z 310.711,A -85,B 0,C 180,E1 -15378.832,E2 -15378.832} C_VEL
LIN {X 0,Y 320.914,Z 316.356,A -85,B 0,C 180,E1 -15380.457,E2 -15380.457} C_VEL
LIN {X 0,Y 326.056,Z 332.233,A -85,B 0,C 180,E1 -15381.146,E2 -15381.146} C_VEL
LIN {X 0,Y 328.404,Z 345.35,A -85,B 0,C 180,E1 -15381.587,E2 -15381.587} C_VEL
LIN {X 0,Y 326.676,Z 424.029,A -85,B 0,C 180,E1 -15383.322,E2 -15383.322} C_VEL
LIN {X 0,Y 326.126,Z 437.001,A -85,B 0,C 180,E1 -15383.854,E2 -15383.854} C_VEL
LIN {X 0,Y 325.351,Z 450.106,A -85,B 0,C 180,E1 -15384.656,E2 -15384.656} C_VEL
LIN {X 0,Y 324.4,Z 462.417,A -85,B 0,C 180,E1 -15385.699,E2 -15385.699} C_VEL
LIN {X 0,Y 323.367,Z 473.328,A -85,B 0,C 180,E1 -15386.886,E2 -15386.886} C_VEL
LIN {X 0,Y 322.221,Z 483.614,A -85,B 0,C 180,E1 -15388.282,E2 -15388.282} C_VEL
LIN {X 0,Y 320.982,Z 493.67,A -85,B 0,C 180,E1 -15390.001,E2 -15390.001} C_VEL
LIN {X 0,Y 319.967,Z 502.498,A -85,B 0,C 180,E1 -15391.889,E2 -15391.889} C_VEL
LIN {X 0,Y 319.191,Z 509.563,A -85,B 0,C 180,E1 -15393.788,E2 -15393.788} C_VEL
LIN {X 0,Y 318.66,Z 515.201,A -85,B 0,C 180,E1 -15395.697,E2 -15395.697} C_VEL
LIN {X 0,Y 318.239,Z 519.647,A -85,B 0,C 180,E1 -15397.615,E2 -15397.615} C_VEL
LIN {X 0,Y 318.009,Z 522.004,A -85,B 0,C 180,E1 -15398.9,E2 -15398.9} C_VEL
LIN {X 0,Y 317.82,Z 523.931,A -85,B 0,C 180,E1 -15400.19,E2 -15400.19} C_VEL
LIN {X 0,Y 317.758,Z 525.38,A -85,B 0,C 180,E1 -15401.483,E2 -15401.483} C_VEL
LIN {X 0,Y 317.731,Z 526.724,A -85,B 0,C 180,E1 -15403.28,E2 -15403.28} C_VEL
LIN {X 0,Y 317.682,Z 527.272,A -85,B 0,C 180,E1 -15405.396,E2 -15405.396} C_VEL
LIN {X 0,Y 317.782,Z 527.041,A -85,B 0,C 180,E1 -15406.709,E2 -15406.709} C_VEL
LIN {X 0,Y 317.956,Z 526.356,A -85,B 0,C 180,E1 -15408.109,E2 -15408.109} C_VEL
LIN {X 0,Y 318.197,Z 525.361,A -85,B 0,C 180,E1 -15409.349,E2 -15409.349} C_VEL
LIN {X 0,Y 318.491,Z 523.834,A -85,B 0,C 180,E1 -15410.676,E2 -15410.676} C_VEL
LIN {X 0,Y 319.062,Z 521.338,A -85,B 0,C 180,E1 -15412.31,E2 -15412.31} C_VEL
LIN {X 0,Y 319.689,Z 517.945,A -85,B 0,C 180,E1 -15413.998,E2 -15413.998} C_VEL
LIN {X 0,Y 320.772,Z 512.602,A -85,B 0,C 180,E1 -15416.064,E2 -15416.064} C_VEL
LIN {X 0,Y 322.062,Z 506.236,A -85,B 0,C 180,E1 -15417.981,E2 -15417.981} C_VEL
LIN {X 0,Y 323.71,Z 497.891,A -85,B 0,C 180,E1 -15419.957,E2 -15419.957} C_VEL
LIN {X 0,Y 325.224,Z 489.269,A -85,B 0,C 180,E1 -15421.604,E2 -15421.604} C_VEL
LIN {X 0,Y 327.051,Z 479.032,A -85,B 0,C 180,E1 -15423.159,E2 -15423.159} C_VEL
LIN {X 0,Y 328.806,Z 467.823,A -85,B 0,C 180,E1 -15424.501,E2 -15424.501} C_VEL
LIN {X 0,Y 330.179,Z 456.692,A -85,B 0,C 180,E1 -15425.56,E2 -15425.56} C_VEL
LIN {X 0,Y 331.402,Z 444.679,A -85,B 0,C 180,E1 -15426.427,E2 -15426.427} C_VEL
LIN {X 0,Y 332.282,Z 431.751,A -85,B 0,C 180,E1 -15427.095,E2 -15427.095} C_VEL
LIN {X 0,Y 332.871,Z 418.672,A -85,B 0,C 180,E1 -15427.517,E2 -15427.517} C_VEL
LIN {X 0,Y 334.87,Z 347.732,A -85,B 0,C 180,E1 -15429.056,E2 -15429.056} C_VEL
LIN {X 0,Y 333.664,Z 343.739,A -85,B 0,C 180,E1 -15429.272,E2 -15429.272} C_VEL
LIN {X 0,Y 332.688,Z 341.332,A -85,B 0,C 180,E1 -15429.427,E2 -15429.427} C_VEL
LIN {X 0,Y 329.997,Z 336.592,A -85,B 0,C 180,E1 -15429.817,E2 -15429.817} C_VEL
LIN {X 0,Y 324.084,Z 330.02,A -85,B 0,C 180,E1 -15430.603,E2 -15430.603} C_VEL
LIN {X 0,Y 319.102,Z 325.007,A -85,B 0,C 180,E1 -15431.28,E2 -15431.28} C_VEL
LIN {X 0,Y 315.809,Z 320.807,A -85,B 0,C 180,E1 -15431.768,E2 -15431.768} C_VEL
LIN {X 0,Y 314.876,Z 319.253,A -85,B 0,C 180,E1 -15431.919,E2 -15431.919} C_VEL
LIN {X 0,Y 313.855,Z 316.918,A -85,B 0,C 180,E1 -15432.143,E2 -15432.143} C_VEL
LIN {X 0,Y 312.453,Z 311.567,A -85,B 0,C 180,E1 -15434.088,E2 -15434.088} C_VEL
LIN {X 0,Y 312.487,Z 311.563,A -85,B 0,C 180,E1 -15437.919,E2 -15437.919} C_VEL
LIN {X 0,Y 312.508,Z 311.553,A -85,B 0,C 180,E1 -15441.917,E2 -15441.917} C_VEL
LIN {X 0,Y 312.534,Z 311.553,A -85,B 0,C 180,E1 -15444.22,E2 -15444.22} C_VEL
LIN {X 0,Y 312.506,Z 311.555,A -85,B 0,C 180,E1 -15447.334,E2 -15447.334} C_VEL
LIN {X 0,Y 312.554,Z 311.554,A -85,B 0,C 180,E1 -15451.276,E2 -15451.276} C_VEL
LIN {X 0,Y 312.588,Z 311.546,A -85,B 0,C 180,E1 -15454.711,E2 -15454.711} C_VEL
LIN {X 0,Y 312.589,Z 311.541,A -85,B 0,C 180,E1 -15457.529,E2 -15457.529} C_VEL
LIN {X 0,Y 312.64,Z 311.533,A -85,B 0,C 180,E1 -15461.656,E2 -15461.656} C_VEL
LIN {X 0,Y 312.695,Z 311.524,A -85,B 0,C 180,E1 -15465.686,E2 -15465.686} C_VEL
LIN {X 0,Y 312.703,Z 311.524,A -85,B 0,C 180,E1 -15469.642,E2 -15469.642} C_VEL
LIN {X 0,Y 312.874,Z 311.512,A -85,B 0,C 180,E1 -15472.254,E2 -15472.254} C_VEL
LIN {X 0,Y 312.717,Z 311.524,A -85,B 0,C 180,E1 -15474.842,E2 -15474.842} C_VEL
LIN {X 0,Y 312.989,Z 311.494,A -85,B 0,C 180,E1 -15478.713,E2 -15478.713} C_VEL
LIN {X 0,Y 312.989,Z 311.481,A -85,B 0,C 180,E1 -15481.287,E2 -15481.287} C_VEL
LIN {X 0,Y 312.717,Z 311.522,A -85,B 0,C 180,E1 -15485.158,E2 -15485.158} C_VEL
LIN {X 0,Y 312.874,Z 311.505,A -85,B 0,C 180,E1 -15487.746,E2 -15487.746} C_VEL
LIN {X 0,Y 312.67,Z 311.521,A -85,B 0,C 180,E1 -15491.671,E2 -15491.671} C_VEL
LIN {X 0,Y 312.701,Z 311.527,A -85,B 0,C 180,E1 -15494.887,E2 -15494.887} C_VEL
LIN {X 0,Y 312.631,Z 311.54,A -85,B 0,C 180,E1 -15499.236,E2 -15499.236} C_VEL
LIN {X 0,Y 312.528,Z 311.554,A -85,B 0,C 180,E1 -15502.78,E2 -15502.78} C_VEL
LIN {X 0,Y 312.598,Z 311.534,A -85,B 0,C 180,E1 -15505.933,E2 -15505.933} C_VEL
LIN {X 0,Y 312.547,Z 311.542,A -85,B 0,C 180,E1 -15509.65,E2 -15509.65} C_VEL
LIN {X 0,Y 312.521,Z 311.546,A -85,B 0,C 180,E1 -15513.689,E2 -15513.689} C_VEL
LIN {X 0,Y 312.527,Z 311.549,A -85,B 0,C 180,E1 -15517.385,E2 -15517.385} C_VEL
LIN {X 0,Y 312.492,Z 311.555,A -85,B 0,C 180,E1 -15520.709,E2 -15520.709} C_VEL
LIN {X 0,Y 312.453,Z 311.565,A -85,B 0,C 180,E1 -15524.209,E2 -15524.209} C_VEL
LIN {X 0,Y 312.486,Z 311.559,A -85,B 0,C 180,E1 -15527.918,E2 -15527.918} C_VEL
LIN {X 0,Y 312.501,Z 311.547,A -85,B 0,C 180,E1 -15530.971,E2 -15530.971} C_VEL
LIN {X 0,Y 312.535,Z 311.581,A -85,B 0,C 180,E1 -15534.319,E2 -15534.319} C_VEL
LIN {X 0,Y 315.264,Z 322.173,A -85,B 0,C 180,E1 -15537.899,E2 -15537.899} C_VEL
LIN {X 0,Y 317.671,Z 332.697,A -85,B 0,C 180,E1 -15541.22,E2 -15541.22} C_VEL
LIN {X 0,Y 318.563,Z 337.132,A -85,B 0,C 180,E1 -15542.513,E2 -15542.513} C_VEL
LIN {X 0,Y 320.463,Z 342.289,A -85,B 0,C 180,E1 -15542.857,E2 -15542.857} C_VEL
LIN {X 0,Y 325.57,Z 366.153,A -85,B 0,C 180,E1 -15544.009,E2 -15544.009} C_VEL
LIN {X 0,Y 327.883,Z 381.003,A -85,B 0,C 180,E1 -15544.615,E2 -15544.615} C_VEL
LIN {X 0,Y 326.061,Z 445.678,A -85,B 0,C 180,E1 -15546.078,E2 -15546.078} C_VEL
LIN {X 0,Y 325.083,Z 458.867,A -85,B 0,C 180,E1 -15546.593,E2 -15546.593} C_VEL
LIN {X 0,Y 323.753,Z 471.542,A -85,B 0,C 180,E1 -15547.336,E2 -15547.336} C_VEL
LIN {X 0,Y 322.258,Z 482.843,A -85,B 0,C 180,E1 -15548.238,E2 -15548.238} C_VEL
LIN {X 0,Y 320.414,Z 494.5,A -85,B 0,C 180,E1 -15549.454,E2 -15549.454} C_VEL
LIN {X 0,Y 318.514,Z 504.988,A -85,B 0,C 180,E1 -15550.839,E2 -15550.839} C_VEL
LIN {X 0,Y 316.889,Z 513.581,A -85,B 0,C 180,E1 -15552.245,E2 -15552.245} C_VEL
LIN {X 0,Y 315.468,Z 521.515,A -85,B 0,C 180,E1 -15553.83,E2 -15553.83} C_VEL
LIN {X 0,Y 313.933,Z 529.327,A -85,B 0,C 180,E1 -15555.743,E2 -15555.743} C_VEL
LIN {X 0,Y 312.614,Z 535.598,A -85,B 0,C 180,E1 -15557.667,E2 -15557.667} C_VEL
LIN {X 0,Y 311.753,Z 540.614,A -85,B 0,C 180,E1 -15559.609,E2 -15559.609} C_VEL
LIN {X 0,Y 311.192,Z 544.52,A -85,B 0,C 180,E1 -15561.558,E2 -15561.558} C_VEL
LIN {X 0,Y 310.767,Z 548.325,A -85,B 0,C 180,E1 -15564.305,E2 -15564.305} C_VEL
LIN {X 0,Y 310.72,Z 549.795,A -85,B 0,C 180,E1 -15566.108,E2 -15566.108} C_VEL
LIN {X 0,Y 310.7,Z 550.403,A -85,B 0,C 180,E1 -15567.406,E2 -15567.406} C_VEL
LIN {X 0,Y 310.692,Z 550.603,A -85,B 0,C 180,E1 -15568.703,E2 -15568.703} C_VEL
LIN {X 0,Y 310.76,Z 550.381,A -85,B 0,C 180,E1 -15569.999,E2 -15569.999} C_VEL
LIN {X 0,Y 310.722,Z 549.766,A -85,B 0,C 180,E1 -15571.295,E2 -15571.295} C_VEL
LIN {X 0,Y 310.722,Z 548.759,A -85,B 0,C 180,E1 -15572.592,E2 -15572.592} C_VEL
LIN {X 0,Y 310.757,Z 547.328,A -85,B 0,C 180,E1 -15573.889,E2 -15573.889} C_VEL
LIN {X 0,Y 310.823,Z 544.414,A -85,B 0,C 180,E1 -15575.798,E2 -15575.798} C_VEL
LIN {X 0,Y 311.001,Z 540.283,A -85,B 0,C 180,E1 -15577.792,E2 -15577.792} C_VEL
LIN {X 0,Y 311.473,Z 534.021,A -85,B 0,C 180,E1 -15580.07,E2 -15580.07} C_VEL
LIN {X 0,Y 312.103,Z 527.18,A -85,B 0,C 180,E1 -15582.021,E2 -15582.021} C_VEL
LIN {X 0,Y 313.108,Z 518.667,A -85,B 0,C 180,E1 -15583.962,E2 -15583.962} C_VEL
LIN {X 0,Y 314.169,Z 509.876,A -85,B 0,C 180,E1 -15585.57,E2 -15585.57} C_VEL
LIN {X 0,Y 315.34,Z 499.026,A -85,B 0,C 180,E1 -15587.175,E2 -15587.175} C_VEL
LIN {X 0,Y 316.485,Z 488.201,A -85,B 0,C 180,E1 -15588.447,E2 -15588.447} C_VEL
LIN {X 0,Y 317.729,Z 476.049,A -85,B 0,C 180,E1 -15589.544,E2 -15589.544} C_VEL
LIN {X 0,Y 318.751,Z 463.348,A -85,B 0,C 180,E1 -15590.403,E2 -15590.403} C_VEL
LIN {X 0,Y 319.537,Z 450.963,A -85,B 0,C 180,E1 -15590.982,E2 -15590.982} C_VEL
LIN {X 0,Y 320.008,Z 435.165,A -85,B 0,C 180,E1 -15591.413,E2 -15591.413} C_VEL
LIN {X 0,Y 321.017,Z 378.328,A -85,B 0,C 180,E1 -15592.68,E2 -15592.68} C_VEL
LIN {X 0,Y 315.565,Z 337.853,A -85,B 0,C 180,E1 -15593.981,E2 -15593.981} C_VEL
LIN {X 0,Y 316.289,Z 331.198,A -85,B 0,C 180,E1 -15595.675,E2 -15595.675} C_VEL
LIN {X 0,Y 314.962,Z 322.944,A -85,B 0,C 180,E1 -15597.941,E2 -15597.941} C_VEL
LIN {X 0,Y 312.514,Z 311.559,A -85,B 0,C 180,E1 -15601.218,E2 -15601.218} C_VEL
LIN {X 0,Y 312.503,Z 311.56,A -85,B 0,C 180,E1 -15604.209,E2 -15604.209} C_VEL
LIN {X 0,Y 312.53,Z 311.555,A -85,B 0,C 180,E1 -15608.088,E2 -15608.088} C_VEL
LIN {X 0,Y 312.479,Z 311.56,A -85,B 0,C 180,E1 -15612.08,E2 -15612.08} C_VEL
LIN {X 0,Y 312.453,Z 311.563,A -85,B 0,C 180,E1 -15616.034,E2 -15616.034} C_VEL
LIN {X 0,Y 312.484,Z 311.557,A -85,B 0,C 180,E1 -15619.29,E2 -15619.29} C_VEL
LIN {X 0,Y 312.532,Z 311.556,A -85,B 0,C 180,E1 -15622.616,E2 -15622.616} C_VEL
LIN {X 0,Y 312.514,Z 311.555,A -85,B 0,C 180,E1 -15626.31,E2 -15626.31} C_VEL
LIN {X 0,Y 312.54,Z 311.551,A -85,B 0,C 180,E1 -15630.349,E2 -15630.349} C_VEL
LIN {X 0,Y 312.595,Z 311.543,A -85,B 0,C 180,E1 -15634.064,E2 -15634.064} C_VEL
LIN {X 0,Y 312.579,Z 311.547,A -85,B 0,C 180,E1 -15637.528,E2 -15637.528} C_VEL
LIN {X 0,Y 312.63,Z 311.537,A -85,B 0,C 180,E1 -15641.656,E2 -15641.656} C_VEL
LIN {X 0,Y 312.685,Z 311.534,A -85,B 0,C 180,E1 -15645.686,E2 -15645.686} C_VEL
LIN {X 0,Y 312.693,Z 311.534,A -85,B 0,C 180,E1 -15649.642,E2 -15649.642} C_VEL
LIN {X 0,Y 312.863,Z 311.507,A -85,B 0,C 180,E1 -15652.254,E2 -15652.254} C_VEL
LIN {X 0,Y 312.709,Z 311.525,A -85,B 0,C 180,E1 -15654.842,E2 -15654.842} C_VEL
LIN {X 0,Y 312.982,Z 311.495,A -85,B 0,C 180,E1 -15658.713,E2 -15658.713} C_VEL
LIN {X 0,Y 312.982,Z 311.497,A -85,B 0,C 180,E1 -15661.287,E2 -15661.287} C_VEL
LIN {X 0,Y 312.698,Z 311.527,A -85,B 0,C 180,E1 -15665.158,E2 -15665.158} C_VEL
LIN {X 0,Y 312.808,Z 311.516,A -85,B 0,C 180,E1 -15667.747,E2 -15667.747} C_VEL
LIN {X 0,Y 312.66,Z 311.538,A -85,B 0,C 180,E1 -15671.672,E2 -15671.672} C_VEL
LIN {X 0,Y 312.692,Z 311.53,A -85,B 0,C 180,E1 -15674.888,E2 -15674.888} C_VEL
LIN {X 0,Y 312.622,Z 311.54,A -85,B 0,C 180,E1 -15679.237,E2 -15679.237} C_VEL
LIN {X 0,Y 312.518,Z 311.554,A -85,B 0,C 180,E1 -15682.781,E2 -15682.781} C_VEL
LIN {X 0,Y 312.595,Z 311.545,A -85,B 0,C 180,E1 -15685.936,E2 -15685.936} C_VEL
LIN {X 0,Y 312.538,Z 311.55,A -85,B 0,C 180,E1 -15689.651,E2 -15689.651} C_VEL
LIN {X 0,Y 312.513,Z 311.552,A -85,B 0,C 180,E1 -15693.69,E2 -15693.69} C_VEL
LIN {X 0,Y 312.507,Z 311.554,A -85,B 0,C 180,E1 -15697.388,E2 -15697.388} C_VEL
LIN {X 0,Y 312.435,Z 311.568,A -85,B 0,C 180,E1 -15700.718,E2 -15700.718} C_VEL
LIN {X 0,Y 312.446,Z 311.561,A -85,B 0,C 180,E1 -15704.211,E2 -15704.211} C_VEL
LIN {X 0,Y 312.45,Z 311.561,A -85,B 0,C 180,E1 -15707.926,E2 -15707.926} C_VEL
LIN {X 0,Y 312.48,Z 311.558,A -85,B 0,C 180,E1 -15711.924,E2 -15711.924} C_VEL
LIN {X 0,Y 312.528,Z 311.552,A -85,B 0,C 180,E1 -15714.221,E2 -15714.221} C_VEL
LIN {X 0,Y 312.498,Z 311.56,A -85,B 0,C 180,E1 -15717.335,E2 -15717.335} C_VEL
LIN {X 0,Y 312.503,Z 311.56,A -85,B 0,C 180,E1 -15721.294,E2 -15721.294} C_VEL
LIN {X 0,Y 312.545,Z 311.551,A -85,B 0,C 180,E1 -15724.709,E2 -15724.709} C_VEL
LIN {X 0,Y 312.525,Z 311.552,A -85,B 0,C 180,E1 -15728.913,E2 -15728.913} C_VEL
LIN {X 0,Y 312.582,Z 311.55,A -85,B 0,C 180,E1 -15731.654,E2 -15731.654} C_VEL
LIN {X 0,Y 312.686,Z 311.537,A -85,B 0,C 180,E1 -15735.687,E2 -15735.687} C_VEL
LIN {X 0,Y 312.692,Z 311.634,A -85,B 0,C 180,E1 -15738.536,E2 -15738.536} C_VEL
LIN {X 0,Y 313.686,Z 316.333,A -85,B 0,C 180,E1 -15739.973,E2 -15739.973} C_VEL
LIN {X 0,Y 319.5,Z 334.006,A -85,B 0,C 180,E1 -15740.784,E2 -15740.784} C_VEL
LIN {X 0,Y 321.692,Z 347.127,A -85,B 0,C 180,E1 -15741.227,E2 -15741.227} C_VEL
LIN {X 0,Y 319.929,Z 423.708,A -85,B 0,C 180,E1 -15742.943,E2 -15742.943} C_VEL
LIN {X 0,Y 319.337,Z 436.885,A -85,B 0,C 180,E1 -15743.485,E2 -15743.485} C_VEL
LIN {X 0,Y 318.53,Z 450.102,A -85,B 0,C 180,E1 -15744.303,E2 -15744.303} C_VEL
LIN {X 0,Y 317.567,Z 462.367,A -85,B 0,C 180,E1 -15745.356,E2 -15745.356} C_VEL
LIN {X 0,Y 316.434,Z 474.073,A -85,B 0,C 180,E1 -15746.659,E2 -15746.659} C_VEL
LIN {X 0,Y 315.232,Z 484.263,A -85,B 0,C 180,E1 -15748.085,E2 -15748.085} C_VEL
LIN {X 0,Y 314.089,Z 493.426,A -85,B 0,C 180,E1 -15749.68,E2 -15749.68} C_VEL
LIN {X 0,Y 312.994,Z 502.347,A -85,B 0,C 180,E1 -15751.609,E2 -15751.609} C_VEL
LIN {X 0,Y 312.181,Z 509.514,A -85,B 0,C 180,E1 -15753.55,E2 -15753.55} C_VEL
LIN {X 0,Y 311.654,Z 514.356,A -85,B 0,C 180,E1 -15755.176,E2 -15755.176} C_VEL
LIN {X 0,Y 311.276,Z 518.907,A -85,B 0,C 180,E1 -15757.069,E2 -15757.069} C_VEL
LIN {X 0,Y 310.877,Z 522.65,A -85,B 0,C 180,E1 -15759.106,E2 -15759.106} C_VEL
LIN {X 0,Y 310.701,Z 524.476,A -85,B 0,C 180,E1 -15760.426,E2 -15760.426} C_VEL
